(* IEC 61131-3 sources: TA/Tests/RetainTest/Man (part 21) *)

    RETAINTEST_AUTO_STRUCTUREARRAYARRAY.ARRAYARRAY_LREAL[2][0] := RETAINTEST_AUTO_STRUCTUREARRAYARRAY.ARRAYARRAY_LREAL[2][0] + 1.1;
    RETAINTEST_AUTO_STRUCTUREARRAYARRAY.ARRAYARRAY_LREAL[2][1] := RETAINTEST_AUTO_STRUCTUREARRAYARRAY.ARRAYARRAY_LREAL[2][1] + 1.1;
    RETAINTEST_AUTO_STRUCTUREARRAYARRAY.ARRAYARRAY_LREAL[2][2] := RETAINTEST_AUTO_STRUCTUREARRAYARRAY.ARRAYARRAY_LREAL[2][2] + 1.1;
    RETAINTEST_AUTO_STRUCTUREARRAYARRAY.ARRAYARRAY_LREAL[2][3] := RETAINTEST_AUTO_STRUCTUREARRAYARRAY.ARRAYARRAY_LREAL[2][3] + 1.1;
    RETAINTEST_AUTO_STRUCTUREARRAYARRAY.ARRAYARRAY_LREAL[2][4] := RETAINTEST_AUTO_STRUCTUREARRAYARRAY.ARRAYARRAY_LREAL[2][4] + 1.1;
    RETAINTEST_AUTO_STRUCTUREARRAYARRAY.ARRAYARRAY_LREAL[2][5] := RETAINTEST_AUTO_STRUCTUREARRAYARRAY.ARRAYARRAY_LREAL[2][5] + 1.1;
    RETAINTEST_AUTO_STRUCTUREARRAYARRAY.ARRAYARRAY_LREAL[2][6] := RETAINTEST_AUTO_STRUCTUREARRAYARRAY.ARRAYARRAY_LREAL[2][6] + 1.1;
    RETAINTEST_AUTO_STRUCTUREARRAYARRAY.ARRAYARRAY_LREAL[2][7] := RETAINTEST_AUTO_STRUCTUREARRAYARRAY.ARRAYARRAY_LREAL[2][7] + 1.1;
    RETAINTEST_AUTO_STRUCTUREARRAYARRAY.ARRAYARRAY_LREAL[2][8] := RETAINTEST_AUTO_STRUCTUREARRAYARRAY.ARRAYARRAY_LREAL[2][8] + 1.1;
    RETAINTEST_AUTO_STRUCTUREARRAYARRAY.ARRAYARRAY_LREAL[2][9] := RETAINTEST_AUTO_STRUCTUREARRAYARRAY.ARRAYARRAY_LREAL[2][9] + 1.1;

    RETAINTEST_AUTO_STRUCTUREARRAYARRAY.ARRAYARRAY_LREAL[3][0] := RETAINTEST_AUTO_STRUCTUREARRAYARRAY.ARRAYARRAY_LREAL[3][0] + 1.1;
    RETAINTEST_AUTO_STRUCTUREARRAYARRAY.ARRAYARRAY_LREAL[3][1] := RETAINTEST_AUTO_STRUCTUREARRAYARRAY.ARRAYARRAY_LREAL[3][1] + 1.1;
    RETAINTEST_AUTO_STRUCTUREARRAYARRAY.ARRAYARRAY_LREAL[3][2] := RETAINTEST_AUTO_STRUCTUREARRAYARRAY.ARRAYARRAY_LREAL[3][2] + 1.1;
    RETAINTEST_AUTO_STRUCTUREARRAYARRAY.ARRAYARRAY_LREAL[3][3] := RETAINTEST_AUTO_STRUCTUREARRAYARRAY.ARRAYARRAY_LREAL[3][3] + 1.1;
    RETAINTEST_AUTO_STRUCTUREARRAYARRAY.ARRAYARRAY_LREAL[3][4] := RETAINTEST_AUTO_STRUCTUREARRAYARRAY.ARRAYARRAY_LREAL[3][4] + 1.1;
    RETAINTEST_AUTO_STRUCTUREARRAYARRAY.ARRAYARRAY_LREAL[3][5] := RETAINTEST_AUTO_STRUCTUREARRAYARRAY.ARRAYARRAY_LREAL[3][5] + 1.1;
    RETAINTEST_AUTO_STRUCTUREARRAYARRAY.ARRAYARRAY_LREAL[3][6] := RETAINTEST_AUTO_STRUCTUREARRAYARRAY.ARRAYARRAY_LREAL[3][6] + 1.1;
    RETAINTEST_AUTO_STRUCTUREARRAYARRAY.ARRAYARRAY_LREAL[3][7] := RETAINTEST_AUTO_STRUCTUREARRAYARRAY.ARRAYARRAY_LREAL[3][7] + 1.1;
    RETAINTEST_AUTO_STRUCTUREARRAYARRAY.ARRAYARRAY_LREAL[3][8] := RETAINTEST_AUTO_STRUCTUREARRAYARRAY.ARRAYARRAY_LREAL[3][8] + 1.1;
    RETAINTEST_AUTO_STRUCTUREARRAYARRAY.ARRAYARRAY_LREAL[3][9] := RETAINTEST_AUTO_STRUCTUREARRAYARRAY.ARRAYARRAY_LREAL[3][9] + 1.1;

    RETAINTEST_AUTO_STRUCTUREARRAYARRAY.ARRAYARRAY_LREAL[4][0] := RETAINTEST_AUTO_STRUCTUREARRAYARRAY.ARRAYARRAY_LREAL[4][0] + 1.1;
    RETAINTEST_AUTO_STRUCTUREARRAYARRAY.ARRAYARRAY_LREAL[4][1] := RETAINTEST_AUTO_STRUCTUREARRAYARRAY.ARRAYARRAY_LREAL[4][1] + 1.1;
    RETAINTEST_AUTO_STRUCTUREARRAYARRAY.ARRAYARRAY_LREAL[4][2] := RETAINTEST_AUTO_STRUCTUREARRAYARRAY.ARRAYARRAY_LREAL[4][2] + 1.1;
    RETAINTEST_AUTO_STRUCTUREARRAYARRAY.ARRAYARRAY_LREAL[4][3] := RETAINTEST_AUTO_STRUCTUREARRAYARRAY.ARRAYARRAY_LREAL[4][3] + 1.1;
    RETAINTEST_AUTO_STRUCTUREARRAYARRAY.ARRAYARRAY_LREAL[4][4] := RETAINTEST_AUTO_STRUCTUREARRAYARRAY.ARRAYARRAY_LREAL[4][4] + 1.1;
    RETAINTEST_AUTO_STRUCTUREARRAYARRAY.ARRAYARRAY_LREAL[4][5] := RETAINTEST_AUTO_STRUCTUREARRAYARRAY.ARRAYARRAY_LREAL[4][5] + 1.1;
    RETAINTEST_AUTO_STRUCTUREARRAYARRAY.ARRAYARRAY_LREAL[4][6] := RETAINTEST_AUTO_STRUCTUREARRAYARRAY.ARRAYARRAY_LREAL[4][6] + 1.1;
    RETAINTEST_AUTO_STRUCTUREARRAYARRAY.ARRAYARRAY_LREAL[4][7] := RETAINTEST_AUTO_STRUCTUREARRAYARRAY.ARRAYARRAY_LREAL[4][7] + 1.1;
    RETAINTEST_AUTO_STRUCTUREARRAYARRAY.ARRAYARRAY_LREAL[4][8] := RETAINTEST_AUTO_STRUCTUREARRAYARRAY.ARRAYARRAY_LREAL[4][8] + 1.1;
    RETAINTEST_AUTO_STRUCTUREARRAYARRAY.ARRAYARRAY_LREAL[4][9] := RETAINTEST_AUTO_STRUCTUREARRAYARRAY.ARRAYARRAY_LREAL[4][9] + 1.1;

    RETAINTEST_AUTO_STRUCTUREARRAYARRAY.ARRAYARRAY_LREAL[5][0] := RETAINTEST_AUTO_STRUCTUREARRAYARRAY.ARRAYARRAY_LREAL[5][0] + 1.1;
    RETAINTEST_AUTO_STRUCTUREARRAYARRAY.ARRAYARRAY_LREAL[5][1] := RETAINTEST_AUTO_STRUCTUREARRAYARRAY.ARRAYARRAY_LREAL[5][1] + 1.1;
    RETAINTEST_AUTO_STRUCTUREARRAYARRAY.ARRAYARRAY_LREAL[5][2] := RETAINTEST_AUTO_STRUCTUREARRAYARRAY.ARRAYARRAY_LREAL[5][2] + 1.1;
    RETAINTEST_AUTO_STRUCTUREARRAYARRAY.ARRAYARRAY_LREAL[5][3] := RETAINTEST_AUTO_STRUCTUREARRAYARRAY.ARRAYARRAY_LREAL[5][3] + 1.1;
    RETAINTEST_AUTO_STRUCTUREARRAYARRAY.ARRAYARRAY_LREAL[5][4] := RETAINTEST_AUTO_STRUCTUREARRAYARRAY.ARRAYARRAY_LREAL[5][4] + 1.1;
    RETAINTEST_AUTO_STRUCTUREARRAYARRAY.ARRAYARRAY_LREAL[5][5] := RETAINTEST_AUTO_STRUCTUREARRAYARRAY.ARRAYARRAY_LREAL[5][5] + 1.1;
    RETAINTEST_AUTO_STRUCTUREARRAYARRAY.ARRAYARRAY_LREAL[5][6] := RETAINTEST_AUTO_STRUCTUREARRAYARRAY.ARRAYARRAY_LREAL[5][6] + 1.1;
    RETAINTEST_AUTO_STRUCTUREARRAYARRAY.ARRAYARRAY_LREAL[5][7] := RETAINTEST_AUTO_STRUCTUREARRAYARRAY.ARRAYARRAY_LREAL[5][7] + 1.1;
    RETAINTEST_AUTO_STRUCTUREARRAYARRAY.ARRAYARRAY_LREAL[5][8] := RETAINTEST_AUTO_STRUCTUREARRAYARRAY.ARRAYARRAY_LREAL[5][8] + 1.1;
    RETAINTEST_AUTO_STRUCTUREARRAYARRAY.ARRAYARRAY_LREAL[5][9] := RETAINTEST_AUTO_STRUCTUREARRAYARRAY.ARRAYARRAY_LREAL[5][9] + 1.1;

    RETAINTEST_AUTO_STRUCTUREARRAYARRAY.ARRAYARRAY_LREAL[6][0] := RETAINTEST_AUTO_STRUCTUREARRAYARRAY.ARRAYARRAY_LREAL[6][0] + 1.1;
    RETAINTEST_AUTO_STRUCTUREARRAYARRAY.ARRAYARRAY_LREAL[6][1] := RETAINTEST_AUTO_STRUCTUREARRAYARRAY.ARRAYARRAY_LREAL[6][1] + 1.1;
    RETAINTEST_AUTO_STRUCTUREARRAYARRAY.ARRAYARRAY_LREAL[6][2] := RETAINTEST_AUTO_STRUCTUREARRAYARRAY.ARRAYARRAY_LREAL[6][2] + 1.1;
    RETAINTEST_AUTO_STRUCTUREARRAYARRAY.ARRAYARRAY_LREAL[6][3] := RETAINTEST_AUTO_STRUCTUREARRAYARRAY.ARRAYARRAY_LREAL[6][3] + 1.1;
    RETAINTEST_AUTO_STRUCTUREARRAYARRAY.ARRAYARRAY_LREAL[6][4] := RETAINTEST_AUTO_STRUCTUREARRAYARRAY.ARRAYARRAY_LREAL[6][4] + 1.1;
    RETAINTEST_AUTO_STRUCTUREARRAYARRAY.ARRAYARRAY_LREAL[6][5] := RETAINTEST_AUTO_STRUCTUREARRAYARRAY.ARRAYARRAY_LREAL[6][5] + 1.1;
    RETAINTEST_AUTO_STRUCTUREARRAYARRAY.ARRAYARRAY_LREAL[6][6] := RETAINTEST_AUTO_STRUCTUREARRAYARRAY.ARRAYARRAY_LREAL[6][6] + 1.1;
    RETAINTEST_AUTO_STRUCTUREARRAYARRAY.ARRAYARRAY_LREAL[6][7] := RETAINTEST_AUTO_STRUCTUREARRAYARRAY.ARRAYARRAY_LREAL[6][7] + 1.1;
    RETAINTEST_AUTO_STRUCTUREARRAYARRAY.ARRAYARRAY_LREAL[6][8] := RETAINTEST_AUTO_STRUCTUREARRAYARRAY.ARRAYARRAY_LREAL[6][8] + 1.1;
    RETAINTEST_AUTO_STRUCTUREARRAYARRAY.ARRAYARRAY_LREAL[6][9] := RETAINTEST_AUTO_STRUCTUREARRAYARRAY.ARRAYARRAY_LREAL[6][9] + 1.1;

    RETAINTEST_AUTO_STRUCTUREARRAYARRAY.ARRAYARRAY_LREAL[7][0] := RETAINTEST_AUTO_STRUCTUREARRAYARRAY.ARRAYARRAY_LREAL[6][0];
    RETAINTEST_AUTO_STRUCTUREARRAYARRAY.ARRAYARRAY_LREAL[7][1] := RETAINTEST_AUTO_STRUCTUREARRAYARRAY.ARRAYARRAY_LREAL[6][1];
    RETAINTEST_AUTO_STRUCTUREARRAYARRAY.ARRAYARRAY_LREAL[7][2] := RETAINTEST_AUTO_STRUCTUREARRAYARRAY.ARRAYARRAY_LREAL[6][2];
    RETAINTEST_AUTO_STRUCTUREARRAYARRAY.ARRAYARRAY_LREAL[7][3] := RETAINTEST_AUTO_STRUCTUREARRAYARRAY.ARRAYARRAY_LREAL[6][3];
    RETAINTEST_AUTO_STRUCTUREARRAYARRAY.ARRAYARRAY_LREAL[7][4] := RETAINTEST_AUTO_STRUCTUREARRAYARRAY.ARRAYARRAY_LREAL[6][4];
    RETAINTEST_AUTO_STRUCTUREARRAYARRAY.ARRAYARRAY_LREAL[7][5] := RETAINTEST_AUTO_STRUCTUREARRAYARRAY.ARRAYARRAY_LREAL[6][5];
    RETAINTEST_AUTO_STRUCTUREARRAYARRAY.ARRAYARRAY_LREAL[7][6] := RETAINTEST_AUTO_STRUCTUREARRAYARRAY.ARRAYARRAY_LREAL[6][6];
    RETAINTEST_AUTO_STRUCTUREARRAYARRAY.ARRAYARRAY_LREAL[7][7] := RETAINTEST_AUTO_STRUCTUREARRAYARRAY.ARRAYARRAY_LREAL[6][7];
    RETAINTEST_AUTO_STRUCTUREARRAYARRAY.ARRAYARRAY_LREAL[7][8] := RETAINTEST_AUTO_STRUCTUREARRAYARRAY.ARRAYARRAY_LREAL[6][8];
    RETAINTEST_AUTO_STRUCTUREARRAYARRAY.ARRAYARRAY_LREAL[7][9] := RETAINTEST_AUTO_STRUCTUREARRAYARRAY.ARRAYARRAY_LREAL[6][9];

    RETAINTEST_AUTO_STRUCTUREARRAYARRAY.ARRAYARRAY_LWORD[0][0] := RETAINTEST_AUTO_STRUCTUREARRAYARRAY.ARRAYARRAY_LWORD[0][0] + 1;
    RETAINTEST_AUTO_STRUCTUREARRAYARRAY.ARRAYARRAY_LWORD[0][1] := RETAINTEST_AUTO_STRUCTUREARRAYARRAY.ARRAYARRAY_LWORD[0][1] + 1;
    RETAINTEST_AUTO_STRUCTUREARRAYARRAY.ARRAYARRAY_LWORD[0][2] := RETAINTEST_AUTO_STRUCTUREARRAYARRAY.ARRAYARRAY_LWORD[0][2] + 1;
    RETAINTEST_AUTO_STRUCTUREARRAYARRAY.ARRAYARRAY_LWORD[0][3] := RETAINTEST_AUTO_STRUCTUREARRAYARRAY.ARRAYARRAY_LWORD[0][3] + 1;
    RETAINTEST_AUTO_STRUCTUREARRAYARRAY.ARRAYARRAY_LWORD[0][4] := RETAINTEST_AUTO_STRUCTUREARRAYARRAY.ARRAYARRAY_LWORD[0][4] + 1;
    RETAINTEST_AUTO_STRUCTUREARRAYARRAY.ARRAYARRAY_LWORD[0][5] := RETAINTEST_AUTO_STRUCTUREARRAYARRAY.ARRAYARRAY_LWORD[0][5] + 1;
    RETAINTEST_AUTO_STRUCTUREARRAYARRAY.ARRAYARRAY_LWORD[0][6] := RETAINTEST_AUTO_STRUCTUREARRAYARRAY.ARRAYARRAY_LWORD[0][6] + 1;
    RETAINTEST_AUTO_STRUCTUREARRAYARRAY.ARRAYARRAY_LWORD[0][7] := RETAINTEST_AUTO_STRUCTUREARRAYARRAY.ARRAYARRAY_LWORD[0][7] + 1;
    RETAINTEST_AUTO_STRUCTUREARRAYARRAY.ARRAYARRAY_LWORD[0][8] := RETAINTEST_AUTO_STRUCTUREARRAYARRAY.ARRAYARRAY_LWORD[0][6];
    RETAINTEST_AUTO_STRUCTUREARRAYARRAY.ARRAYARRAY_LWORD[0][9] := RETAINTEST_AUTO_STRUCTUREARRAYARRAY.ARRAYARRAY_LWORD[0][7];

    RETAINTEST_AUTO_STRUCTUREARRAYARRAY.ARRAYARRAY_LWORD[1][0] := RETAINTEST_AUTO_STRUCTUREARRAYARRAY.ARRAYARRAY_LWORD[1][0] + 1;
    RETAINTEST_AUTO_STRUCTUREARRAYARRAY.ARRAYARRAY_LWORD[1][1] := RETAINTEST_AUTO_STRUCTUREARRAYARRAY.ARRAYARRAY_LWORD[1][1] + 1;
    RETAINTEST_AUTO_STRUCTUREARRAYARRAY.ARRAYARRAY_LWORD[1][2] := RETAINTEST_AUTO_STRUCTUREARRAYARRAY.ARRAYARRAY_LWORD[1][2] + 1;
    RETAINTEST_AUTO_STRUCTUREARRAYARRAY.ARRAYARRAY_LWORD[1][3] := RETAINTEST_AUTO_STRUCTUREARRAYARRAY.ARRAYARRAY_LWORD[1][3] + 1;
    RETAINTEST_AUTO_STRUCTUREARRAYARRAY.ARRAYARRAY_LWORD[1][4] := RETAINTEST_AUTO_STRUCTUREARRAYARRAY.ARRAYARRAY_LWORD[1][4] + 1;
    RETAINTEST_AUTO_STRUCTUREARRAYARRAY.ARRAYARRAY_LWORD[1][5] := RETAINTEST_AUTO_STRUCTUREARRAYARRAY.ARRAYARRAY_LWORD[1][5] + 1;
    RETAINTEST_AUTO_STRUCTUREARRAYARRAY.ARRAYARRAY_LWORD[1][6] := RETAINTEST_AUTO_STRUCTUREARRAYARRAY.ARRAYARRAY_LWORD[1][6] + 1;
    RETAINTEST_AUTO_STRUCTUREARRAYARRAY.ARRAYARRAY_LWORD[1][7] := RETAINTEST_AUTO_STRUCTUREARRAYARRAY.ARRAYARRAY_LWORD[1][7] + 1;
    RETAINTEST_AUTO_STRUCTUREARRAYARRAY.ARRAYARRAY_LWORD[1][8] := RETAINTEST_AUTO_STRUCTUREARRAYARRAY.ARRAYARRAY_LWORD[1][6];
    RETAINTEST_AUTO_STRUCTUREARRAYARRAY.ARRAYARRAY_LWORD[1][9] := RETAINTEST_AUTO_STRUCTUREARRAYARRAY.ARRAYARRAY_LWORD[1][7];

    RETAINTEST_AUTO_STRUCTUREARRAYARRAY.ARRAYARRAY_LWORD[2][0] := RETAINTEST_AUTO_STRUCTUREARRAYARRAY.ARRAYARRAY_LWORD[2][0] + 1;
    RETAINTEST_AUTO_STRUCTUREARRAYARRAY.ARRAYARRAY_LWORD[2][1] := RETAINTEST_AUTO_STRUCTUREARRAYARRAY.ARRAYARRAY_LWORD[2][1] + 1;
    RETAINTEST_AUTO_STRUCTUREARRAYARRAY.ARRAYARRAY_LWORD[2][2] := RETAINTEST_AUTO_STRUCTUREARRAYARRAY.ARRAYARRAY_LWORD[2][2] + 1;
    RETAINTEST_AUTO_STRUCTUREARRAYARRAY.ARRAYARRAY_LWORD[2][3] := RETAINTEST_AUTO_STRUCTUREARRAYARRAY.ARRAYARRAY_LWORD[2][3] + 1;
    RETAINTEST_AUTO_STRUCTUREARRAYARRAY.ARRAYARRAY_LWORD[2][4] := RETAINTEST_AUTO_STRUCTUREARRAYARRAY.ARRAYARRAY_LWORD[2][4] + 1;
    RETAINTEST_AUTO_STRUCTUREARRAYARRAY.ARRAYARRAY_LWORD[2][5] := RETAINTEST_AUTO_STRUCTUREARRAYARRAY.ARRAYARRAY_LWORD[2][5] + 1;
    RETAINTEST_AUTO_STRUCTUREARRAYARRAY.ARRAYARRAY_LWORD[2][6] := RETAINTEST_AUTO_STRUCTUREARRAYARRAY.ARRAYARRAY_LWORD[2][6] + 1;
    RETAINTEST_AUTO_STRUCTUREARRAYARRAY.ARRAYARRAY_LWORD[2][7] := RETAINTEST_AUTO_STRUCTUREARRAYARRAY.ARRAYARRAY_LWORD[2][7] + 1;
    RETAINTEST_AUTO_STRUCTUREARRAYARRAY.ARRAYARRAY_LWORD[2][8] := RETAINTEST_AUTO_STRUCTUREARRAYARRAY.ARRAYARRAY_LWORD[2][8] + 1;
    RETAINTEST_AUTO_STRUCTUREARRAYARRAY.ARRAYARRAY_LWORD[2][9] := RETAINTEST_AUTO_STRUCTUREARRAYARRAY.ARRAYARRAY_LWORD[2][9] + 1;

    RETAINTEST_AUTO_STRUCTUREARRAYARRAY.ARRAYARRAY_LWORD[3][0] := RETAINTEST_AUTO_STRUCTUREARRAYARRAY.ARRAYARRAY_LWORD[3][0] + 1;
    RETAINTEST_AUTO_STRUCTUREARRAYARRAY.ARRAYARRAY_LWORD[3][1] := RETAINTEST_AUTO_STRUCTUREARRAYARRAY.ARRAYARRAY_LWORD[3][1] + 1;
    RETAINTEST_AUTO_STRUCTUREARRAYARRAY.ARRAYARRAY_LWORD[3][2] := RETAINTEST_AUTO_STRUCTUREARRAYARRAY.ARRAYARRAY_LWORD[3][2] + 1;
    RETAINTEST_AUTO_STRUCTUREARRAYARRAY.ARRAYARRAY_LWORD[3][3] := RETAINTEST_AUTO_STRUCTUREARRAYARRAY.ARRAYARRAY_LWORD[3][3] + 1;
    RETAINTEST_AUTO_STRUCTUREARRAYARRAY.ARRAYARRAY_LWORD[3][4] := RETAINTEST_AUTO_STRUCTUREARRAYARRAY.ARRAYARRAY_LWORD[3][4] + 1;
    RETAINTEST_AUTO_STRUCTUREARRAYARRAY.ARRAYARRAY_LWORD[3][5] := RETAINTEST_AUTO_STRUCTUREARRAYARRAY.ARRAYARRAY_LWORD[3][5] + 1;
    RETAINTEST_AUTO_STRUCTUREARRAYARRAY.ARRAYARRAY_LWORD[3][6] := RETAINTEST_AUTO_STRUCTUREARRAYARRAY.ARRAYARRAY_LWORD[3][6] + 1;
    RETAINTEST_AUTO_STRUCTUREARRAYARRAY.ARRAYARRAY_LWORD[3][7] := RETAINTEST_AUTO_STRUCTUREARRAYARRAY.ARRAYARRAY_LWORD[3][7] + 1;
    RETAINTEST_AUTO_STRUCTUREARRAYARRAY.ARRAYARRAY_LWORD[3][8] := RETAINTEST_AUTO_STRUCTUREARRAYARRAY.ARRAYARRAY_LWORD[3][8] + 1;
    RETAINTEST_AUTO_STRUCTUREARRAYARRAY.ARRAYARRAY_LWORD[3][9] := RETAINTEST_AUTO_STRUCTUREARRAYARRAY.ARRAYARRAY_LWORD[3][9] + 1;

    RETAINTEST_AUTO_STRUCTUREARRAYARRAY.ARRAYARRAY_LWORD[4][0] := RETAINTEST_AUTO_STRUCTUREARRAYARRAY.ARRAYARRAY_LWORD[4][0] + 1;
    RETAINTEST_AUTO_STRUCTUREARRAYARRAY.ARRAYARRAY_LWORD[4][1] := RETAINTEST_AUTO_STRUCTUREARRAYARRAY.ARRAYARRAY_LWORD[4][1] + 1;
    RETAINTEST_AUTO_STRUCTUREARRAYARRAY.ARRAYARRAY_LWORD[4][2] := RETAINTEST_AUTO_STRUCTUREARRAYARRAY.ARRAYARRAY_LWORD[4][2] + 1;
    RETAINTEST_AUTO_STRUCTUREARRAYARRAY.ARRAYARRAY_LWORD[4][3] := RETAINTEST_AUTO_STRUCTUREARRAYARRAY.ARRAYARRAY_LWORD[4][3] + 1;
    RETAINTEST_AUTO_STRUCTUREARRAYARRAY.ARRAYARRAY_LWORD[4][4] := RETAINTEST_AUTO_STRUCTUREARRAYARRAY.ARRAYARRAY_LWORD[4][4] + 1;
    RETAINTEST_AUTO_STRUCTUREARRAYARRAY.ARRAYARRAY_LWORD[4][5] := RETAINTEST_AUTO_STRUCTUREARRAYARRAY.ARRAYARRAY_LWORD[4][5] + 1;
    RETAINTEST_AUTO_STRUCTUREARRAYARRAY.ARRAYARRAY_LWORD[4][6] := RETAINTEST_AUTO_STRUCTUREARRAYARRAY.ARRAYARRAY_LWORD[4][6] + 1;
    RETAINTEST_AUTO_STRUCTUREARRAYARRAY.ARRAYARRAY_LWORD[4][7] := RETAINTEST_AUTO_STRUCTUREARRAYARRAY.ARRAYARRAY_LWORD[4][7] + 1;
    RETAINTEST_AUTO_STRUCTUREARRAYARRAY.ARRAYARRAY_LWORD[4][8] := RETAINTEST_AUTO_STRUCTUREARRAYARRAY.ARRAYARRAY_LWORD[4][8] + 1;
    RETAINTEST_AUTO_STRUCTUREARRAYARRAY.ARRAYARRAY_LWORD[4][9] := RETAINTEST_AUTO_STRUCTUREARRAYARRAY.ARRAYARRAY_LWORD[4][9] + 1;

    RETAINTEST_AUTO_STRUCTUREARRAYARRAY.ARRAYARRAY_LWORD[5][0] := RETAINTEST_AUTO_STRUCTUREARRAYARRAY.ARRAYARRAY_LWORD[5][0] + 1;
    RETAINTEST_AUTO_STRUCTUREARRAYARRAY.ARRAYARRAY_LWORD[5][1] := RETAINTEST_AUTO_STRUCTUREARRAYARRAY.ARRAYARRAY_LWORD[5][1] + 1;
    RETAINTEST_AUTO_STRUCTUREARRAYARRAY.ARRAYARRAY_LWORD[5][2] := RETAINTEST_AUTO_STRUCTUREARRAYARRAY.ARRAYARRAY_LWORD[5][2] + 1;
    RETAINTEST_AUTO_STRUCTUREARRAYARRAY.ARRAYARRAY_LWORD[5][3] := RETAINTEST_AUTO_STRUCTUREARRAYARRAY.ARRAYARRAY_LWORD[5][3] + 1;
    RETAINTEST_AUTO_STRUCTUREARRAYARRAY.ARRAYARRAY_LWORD[5][4] := RETAINTEST_AUTO_STRUCTUREARRAYARRAY.ARRAYARRAY_LWORD[5][4] + 1;
    RETAINTEST_AUTO_STRUCTUREARRAYARRAY.ARRAYARRAY_LWORD[5][5] := RETAINTEST_AUTO_STRUCTUREARRAYARRAY.ARRAYARRAY_LWORD[5][5] + 1;
    RETAINTEST_AUTO_STRUCTUREARRAYARRAY.ARRAYARRAY_LWORD[5][6] := RETAINTEST_AUTO_STRUCTUREARRAYARRAY.ARRAYARRAY_LWORD[5][6] + 1;
    RETAINTEST_AUTO_STRUCTUREARRAYARRAY.ARRAYARRAY_LWORD[5][7] := RETAINTEST_AUTO_STRUCTUREARRAYARRAY.ARRAYARRAY_LWORD[5][7] + 1;
    RETAINTEST_AUTO_STRUCTUREARRAYARRAY.ARRAYARRAY_LWORD[5][8] := RETAINTEST_AUTO_STRUCTUREARRAYARRAY.ARRAYARRAY_LWORD[5][8] + 1;
    RETAINTEST_AUTO_STRUCTUREARRAYARRAY.ARRAYARRAY_LWORD[5][9] := RETAINTEST_AUTO_STRUCTUREARRAYARRAY.ARRAYARRAY_LWORD[5][9] + 1;

    RETAINTEST_AUTO_STRUCTUREARRAYARRAY.ARRAYARRAY_LWORD[6][0] := RETAINTEST_AUTO_STRUCTUREARRAYARRAY.ARRAYARRAY_LWORD[6][0] + 1;
    RETAINTEST_AUTO_STRUCTUREARRAYARRAY.ARRAYARRAY_LWORD[6][1] := RETAINTEST_AUTO_STRUCTUREARRAYARRAY.ARRAYARRAY_LWORD[6][1] + 1;
    RETAINTEST_AUTO_STRUCTUREARRAYARRAY.ARRAYARRAY_LWORD[6][2] := RETAINTEST_AUTO_STRUCTUREARRAYARRAY.ARRAYARRAY_LWORD[6][2] + 1;
    RETAINTEST_AUTO_STRUCTUREARRAYARRAY.ARRAYARRAY_LWORD[6][3] := RETAINTEST_AUTO_STRUCTUREARRAYARRAY.ARRAYARRAY_LWORD[6][3] + 1;
    RETAINTEST_AUTO_STRUCTUREARRAYARRAY.ARRAYARRAY_LWORD[6][4] := RETAINTEST_AUTO_STRUCTUREARRAYARRAY.ARRAYARRAY_LWORD[6][4] + 1;
    RETAINTEST_AUTO_STRUCTUREARRAYARRAY.ARRAYARRAY_LWORD[6][5] := RETAINTEST_AUTO_STRUCTUREARRAYARRAY.ARRAYARRAY_LWORD[6][5] + 1;
    RETAINTEST_AUTO_STRUCTUREARRAYARRAY.ARRAYARRAY_LWORD[6][6] := RETAINTEST_AUTO_STRUCTUREARRAYARRAY.ARRAYARRAY_LWORD[6][6] + 1;
    RETAINTEST_AUTO_STRUCTUREARRAYARRAY.ARRAYARRAY_LWORD[6][7] := RETAINTEST_AUTO_STRUCTUREARRAYARRAY.ARRAYARRAY_LWORD[6][7] + 1;
    RETAINTEST_AUTO_STRUCTUREARRAYARRAY.ARRAYARRAY_LWORD[6][8] := RETAINTEST_AUTO_STRUCTUREARRAYARRAY.ARRAYARRAY_LWORD[6][8] + 1;
    RETAINTEST_AUTO_STRUCTUREARRAYARRAY.ARRAYARRAY_LWORD[6][9] := RETAINTEST_AUTO_STRUCTUREARRAYARRAY.ARRAYARRAY_LWORD[6][9] + 1;

    RETAINTEST_AUTO_STRUCTUREARRAYARRAY.ARRAYARRAY_LWORD[7][0] := RETAINTEST_AUTO_STRUCTUREARRAYARRAY.ARRAYARRAY_LWORD[6][0];
    RETAINTEST_AUTO_STRUCTUREARRAYARRAY.ARRAYARRAY_LWORD[7][1] := RETAINTEST_AUTO_STRUCTUREARRAYARRAY.ARRAYARRAY_LWORD[6][1];
    RETAINTEST_AUTO_STRUCTUREARRAYARRAY.ARRAYARRAY_LWORD[7][2] := RETAINTEST_AUTO_STRUCTUREARRAYARRAY.ARRAYARRAY_LWORD[6][2];
    RETAINTEST_AUTO_STRUCTUREARRAYARRAY.ARRAYARRAY_LWORD[7][3] := RETAINTEST_AUTO_STRUCTUREARRAYARRAY.ARRAYARRAY_LWORD[6][3];
    RETAINTEST_AUTO_STRUCTUREARRAYARRAY.ARRAYARRAY_LWORD[7][4] := RETAINTEST_AUTO_STRUCTUREARRAYARRAY.ARRAYARRAY_LWORD[6][4];
    RETAINTEST_AUTO_STRUCTUREARRAYARRAY.ARRAYARRAY_LWORD[7][5] := RETAINTEST_AUTO_STRUCTUREARRAYARRAY.ARRAYARRAY_LWORD[6][5];
    RETAINTEST_AUTO_STRUCTUREARRAYARRAY.ARRAYARRAY_LWORD[7][6] := RETAINTEST_AUTO_STRUCTUREARRAYARRAY.ARRAYARRAY_LWORD[6][6];
    RETAINTEST_AUTO_STRUCTUREARRAYARRAY.ARRAYARRAY_LWORD[7][7] := RETAINTEST_AUTO_STRUCTUREARRAYARRAY.ARRAYARRAY_LWORD[6][7];
    RETAINTEST_AUTO_STRUCTUREARRAYARRAY.ARRAYARRAY_LWORD[7][8] := RETAINTEST_AUTO_STRUCTUREARRAYARRAY.ARRAYARRAY_LWORD[6][8];
    RETAINTEST_AUTO_STRUCTUREARRAYARRAY.ARRAYARRAY_LWORD[7][9] := RETAINTEST_AUTO_STRUCTUREARRAYARRAY.ARRAYARRAY_LWORD[6][9];

    RETAINTEST_AUTO_STRUCTUREARRAYARRAY.ARRAYARRAY_REAL[0][0] := RETAINTEST_AUTO_STRUCTUREARRAYARRAY.ARRAYARRAY_REAL[0][0] + 1.1;
    RETAINTEST_AUTO_STRUCTUREARRAYARRAY.ARRAYARRAY_REAL[0][1] := RETAINTEST_AUTO_STRUCTUREARRAYARRAY.ARRAYARRAY_REAL[0][1] + 1.1;
    RETAINTEST_AUTO_STRUCTUREARRAYARRAY.ARRAYARRAY_REAL[0][2] := RETAINTEST_AUTO_STRUCTUREARRAYARRAY.ARRAYARRAY_REAL[0][2] + 1.1;
    RETAINTEST_AUTO_STRUCTUREARRAYARRAY.ARRAYARRAY_REAL[0][3] := RETAINTEST_AUTO_STRUCTUREARRAYARRAY.ARRAYARRAY_REAL[0][3] + 1.1;
    RETAINTEST_AUTO_STRUCTUREARRAYARRAY.ARRAYARRAY_REAL[0][4] := RETAINTEST_AUTO_STRUCTUREARRAYARRAY.ARRAYARRAY_REAL[0][4] + 1.1;
    RETAINTEST_AUTO_STRUCTUREARRAYARRAY.ARRAYARRAY_REAL[0][5] := RETAINTEST_AUTO_STRUCTUREARRAYARRAY.ARRAYARRAY_REAL[0][5] + 1.1;
    RETAINTEST_AUTO_STRUCTUREARRAYARRAY.ARRAYARRAY_REAL[0][6] := RETAINTEST_AUTO_STRUCTUREARRAYARRAY.ARRAYARRAY_REAL[0][6] + 1.1;
    RETAINTEST_AUTO_STRUCTUREARRAYARRAY.ARRAYARRAY_REAL[0][7] := RETAINTEST_AUTO_STRUCTUREARRAYARRAY.ARRAYARRAY_REAL[0][7] + 1.1;
    RETAINTEST_AUTO_STRUCTUREARRAYARRAY.ARRAYARRAY_REAL[0][8] := RETAINTEST_AUTO_STRUCTUREARRAYARRAY.ARRAYARRAY_REAL[0][6];
    RETAINTEST_AUTO_STRUCTUREARRAYARRAY.ARRAYARRAY_REAL[0][9] := RETAINTEST_AUTO_STRUCTUREARRAYARRAY.ARRAYARRAY_REAL[0][7];

    RETAINTEST_AUTO_STRUCTUREARRAYARRAY.ARRAYARRAY_REAL[1][0] := RETAINTEST_AUTO_STRUCTUREARRAYARRAY.ARRAYARRAY_REAL[1][0] + 1.1;
    RETAINTEST_AUTO_STRUCTUREARRAYARRAY.ARRAYARRAY_REAL[1][1] := RETAINTEST_AUTO_STRUCTUREARRAYARRAY.ARRAYARRAY_REAL[1][1] + 1.1;
    RETAINTEST_AUTO_STRUCTUREARRAYARRAY.ARRAYARRAY_REAL[1][2] := RETAINTEST_AUTO_STRUCTUREARRAYARRAY.ARRAYARRAY_REAL[1][2] + 1.1;
    RETAINTEST_AUTO_STRUCTUREARRAYARRAY.ARRAYARRAY_REAL[1][3] := RETAINTEST_AUTO_STRUCTUREARRAYARRAY.ARRAYARRAY_REAL[1][3] + 1.1;
    RETAINTEST_AUTO_STRUCTUREARRAYARRAY.ARRAYARRAY_REAL[1][4] := RETAINTEST_AUTO_STRUCTUREARRAYARRAY.ARRAYARRAY_REAL[1][4] + 1.1;
    RETAINTEST_AUTO_STRUCTUREARRAYARRAY.ARRAYARRAY_REAL[1][5] := RETAINTEST_AUTO_STRUCTUREARRAYARRAY.ARRAYARRAY_REAL[1][5] + 1.1;
    RETAINTEST_AUTO_STRUCTUREARRAYARRAY.ARRAYARRAY_REAL[1][6] := RETAINTEST_AUTO_STRUCTUREARRAYARRAY.ARRAYARRAY_REAL[1][6] + 1.1;
    RETAINTEST_AUTO_STRUCTUREARRAYARRAY.ARRAYARRAY_REAL[1][7] := RETAINTEST_AUTO_STRUCTUREARRAYARRAY.ARRAYARRAY_REAL[1][7] + 1.1;
    RETAINTEST_AUTO_STRUCTUREARRAYARRAY.ARRAYARRAY_REAL[1][8] := RETAINTEST_AUTO_STRUCTUREARRAYARRAY.ARRAYARRAY_REAL[1][6];
    RETAINTEST_AUTO_STRUCTUREARRAYARRAY.ARRAYARRAY_REAL[1][9] := RETAINTEST_AUTO_STRUCTUREARRAYARRAY.ARRAYARRAY_REAL[1][7];

    RETAINTEST_AUTO_STRUCTUREARRAYARRAY.ARRAYARRAY_REAL[2][0] := RETAINTEST_AUTO_STRUCTUREARRAYARRAY.ARRAYARRAY_REAL[2][0] + 1.1;
    RETAINTEST_AUTO_STRUCTUREARRAYARRAY.ARRAYARRAY_REAL[2][1] := RETAINTEST_AUTO_STRUCTUREARRAYARRAY.ARRAYARRAY_REAL[2][1] + 1.1;
    RETAINTEST_AUTO_STRUCTUREARRAYARRAY.ARRAYARRAY_REAL[2][2] := RETAINTEST_AUTO_STRUCTUREARRAYARRAY.ARRAYARRAY_REAL[2][2] + 1.1;
    RETAINTEST_AUTO_STRUCTUREARRAYARRAY.ARRAYARRAY_REAL[2][3] := RETAINTEST_AUTO_STRUCTUREARRAYARRAY.ARRAYARRAY_REAL[2][3] + 1.1;
    RETAINTEST_AUTO_STRUCTUREARRAYARRAY.ARRAYARRAY_REAL[2][4] := RETAINTEST_AUTO_STRUCTUREARRAYARRAY.ARRAYARRAY_REAL[2][4] + 1.1;
    RETAINTEST_AUTO_STRUCTUREARRAYARRAY.ARRAYARRAY_REAL[2][5] := RETAINTEST_AUTO_STRUCTUREARRAYARRAY.ARRAYARRAY_REAL[2][5] + 1.1;
    RETAINTEST_AUTO_STRUCTUREARRAYARRAY.ARRAYARRAY_REAL[2][6] := RETAINTEST_AUTO_STRUCTUREARRAYARRAY.ARRAYARRAY_REAL[2][6] + 1.1;
    RETAINTEST_AUTO_STRUCTUREARRAYARRAY.ARRAYARRAY_REAL[2][7] := RETAINTEST_AUTO_STRUCTUREARRAYARRAY.ARRAYARRAY_REAL[2][7] + 1.1;
    RETAINTEST_AUTO_STRUCTUREARRAYARRAY.ARRAYARRAY_REAL[2][8] := RETAINTEST_AUTO_STRUCTUREARRAYARRAY.ARRAYARRAY_REAL[2][8] + 1.1;
    RETAINTEST_AUTO_STRUCTUREARRAYARRAY.ARRAYARRAY_REAL[2][9] := RETAINTEST_AUTO_STRUCTUREARRAYARRAY.ARRAYARRAY_REAL[2][9] + 1.1;

    RETAINTEST_AUTO_STRUCTUREARRAYARRAY.ARRAYARRAY_REAL[3][0] := RETAINTEST_AUTO_STRUCTUREARRAYARRAY.ARRAYARRAY_REAL[3][0] + 1.1;
    RETAINTEST_AUTO_STRUCTUREARRAYARRAY.ARRAYARRAY_REAL[3][1] := RETAINTEST_AUTO_STRUCTUREARRAYARRAY.ARRAYARRAY_REAL[3][1] + 1.1;
    RETAINTEST_AUTO_STRUCTUREARRAYARRAY.ARRAYARRAY_REAL[3][2] := RETAINTEST_AUTO_STRUCTUREARRAYARRAY.ARRAYARRAY_REAL[3][2] + 1.1;
    RETAINTEST_AUTO_STRUCTUREARRAYARRAY.ARRAYARRAY_REAL[3][3] := RETAINTEST_AUTO_STRUCTUREARRAYARRAY.ARRAYARRAY_REAL[3][3] + 1.1;
    RETAINTEST_AUTO_STRUCTUREARRAYARRAY.ARRAYARRAY_REAL[3][4] := RETAINTEST_AUTO_STRUCTUREARRAYARRAY.ARRAYARRAY_REAL[3][4] + 1.1;
    RETAINTEST_AUTO_STRUCTUREARRAYARRAY.ARRAYARRAY_REAL[3][5] := RETAINTEST_AUTO_STRUCTUREARRAYARRAY.ARRAYARRAY_REAL[3][5] + 1.1;
    RETAINTEST_AUTO_STRUCTUREARRAYARRAY.ARRAYARRAY_REAL[3][6] := RETAINTEST_AUTO_STRUCTUREARRAYARRAY.ARRAYARRAY_REAL[3][6] + 1.1;
    RETAINTEST_AUTO_STRUCTUREARRAYARRAY.ARRAYARRAY_REAL[3][7] := RETAINTEST_AUTO_STRUCTUREARRAYARRAY.ARRAYARRAY_REAL[3][7] + 1.1;
    RETAINTEST_AUTO_STRUCTUREARRAYARRAY.ARRAYARRAY_REAL[3][8] := RETAINTEST_AUTO_STRUCTUREARRAYARRAY.ARRAYARRAY_REAL[3][8] + 1.1;
    RETAINTEST_AUTO_STRUCTUREARRAYARRAY.ARRAYARRAY_REAL[3][9] := RETAINTEST_AUTO_STRUCTUREARRAYARRAY.ARRAYARRAY_REAL[3][9] + 1.1;

    RETAINTEST_AUTO_STRUCTUREARRAYARRAY.ARRAYARRAY_REAL[4][0] := RETAINTEST_AUTO_STRUCTUREARRAYARRAY.ARRAYARRAY_REAL[4][0] + 1.1;
    RETAINTEST_AUTO_STRUCTUREARRAYARRAY.ARRAYARRAY_REAL[4][1] := RETAINTEST_AUTO_STRUCTUREARRAYARRAY.ARRAYARRAY_REAL[4][1] + 1.1;
    RETAINTEST_AUTO_STRUCTUREARRAYARRAY.ARRAYARRAY_REAL[4][2] := RETAINTEST_AUTO_STRUCTUREARRAYARRAY.ARRAYARRAY_REAL[4][2] + 1.1;
    RETAINTEST_AUTO_STRUCTUREARRAYARRAY.ARRAYARRAY_REAL[4][3] := RETAINTEST_AUTO_STRUCTUREARRAYARRAY.ARRAYARRAY_REAL[4][3] + 1.1;
    RETAINTEST_AUTO_STRUCTUREARRAYARRAY.ARRAYARRAY_REAL[4][4] := RETAINTEST_AUTO_STRUCTUREARRAYARRAY.ARRAYARRAY_REAL[4][4] + 1.1;
    RETAINTEST_AUTO_STRUCTUREARRAYARRAY.ARRAYARRAY_REAL[4][5] := RETAINTEST_AUTO_STRUCTUREARRAYARRAY.ARRAYARRAY_REAL[4][5] + 1.1;
    RETAINTEST_AUTO_STRUCTUREARRAYARRAY.ARRAYARRAY_REAL[4][6] := RETAINTEST_AUTO_STRUCTUREARRAYARRAY.ARRAYARRAY_REAL[4][6] + 1.1;
    RETAINTEST_AUTO_STRUCTUREARRAYARRAY.ARRAYARRAY_REAL[4][7] := RETAINTEST_AUTO_STRUCTUREARRAYARRAY.ARRAYARRAY_REAL[4][7] + 1.1;
    RETAINTEST_AUTO_STRUCTUREARRAYARRAY.ARRAYARRAY_REAL[4][8] := RETAINTEST_AUTO_STRUCTUREARRAYARRAY.ARRAYARRAY_REAL[4][8] + 1.1;
    RETAINTEST_AUTO_STRUCTUREARRAYARRAY.ARRAYARRAY_REAL[4][9] := RETAINTEST_AUTO_STRUCTUREARRAYARRAY.ARRAYARRAY_REAL[4][9] + 1.1;

    RETAINTEST_AUTO_STRUCTUREARRAYARRAY.ARRAYARRAY_REAL[5][0] := RETAINTEST_AUTO_STRUCTUREARRAYARRAY.ARRAYARRAY_REAL[5][0] + 1.1;
    RETAINTEST_AUTO_STRUCTUREARRAYARRAY.ARRAYARRAY_REAL[5][1] := RETAINTEST_AUTO_STRUCTUREARRAYARRAY.ARRAYARRAY_REAL[5][1] + 1.1;
    RETAINTEST_AUTO_STRUCTUREARRAYARRAY.ARRAYARRAY_REAL[5][2] := RETAINTEST_AUTO_STRUCTUREARRAYARRAY.ARRAYARRAY_REAL[5][2] + 1.1;
    RETAINTEST_AUTO_STRUCTUREARRAYARRAY.ARRAYARRAY_REAL[5][3] := RETAINTEST_AUTO_STRUCTUREARRAYARRAY.ARRAYARRAY_REAL[5][3] + 1.1;
    RETAINTEST_AUTO_STRUCTUREARRAYARRAY.ARRAYARRAY_REAL[5][4] := RETAINTEST_AUTO_STRUCTUREARRAYARRAY.ARRAYARRAY_REAL[5][4] + 1.1;
    RETAINTEST_AUTO_STRUCTUREARRAYARRAY.ARRAYARRAY_REAL[5][5] := RETAINTEST_AUTO_STRUCTUREARRAYARRAY.ARRAYARRAY_REAL[5][5] + 1.1;
    RETAINTEST_AUTO_STRUCTUREARRAYARRAY.ARRAYARRAY_REAL[5][6] := RETAINTEST_AUTO_STRUCTUREARRAYARRAY.ARRAYARRAY_REAL[5][6] + 1.1;
    RETAINTEST_AUTO_STRUCTUREARRAYARRAY.ARRAYARRAY_REAL[5][7] := RETAINTEST_AUTO_STRUCTUREARRAYARRAY.ARRAYARRAY_REAL[5][7] + 1.1;
    RETAINTEST_AUTO_STRUCTUREARRAYARRAY.ARRAYARRAY_REAL[5][8] := RETAINTEST_AUTO_STRUCTUREARRAYARRAY.ARRAYARRAY_REAL[5][8] + 1.1;
    RETAINTEST_AUTO_STRUCTUREARRAYARRAY.ARRAYARRAY_REAL[5][9] := RETAINTEST_AUTO_STRUCTUREARRAYARRAY.ARRAYARRAY_REAL[5][9] + 1.1;

    RETAINTEST_AUTO_STRUCTUREARRAYARRAY.ARRAYARRAY_REAL[6][0] := RETAINTEST_AUTO_STRUCTUREARRAYARRAY.ARRAYARRAY_REAL[6][0] + 1.1;
    RETAINTEST_AUTO_STRUCTUREARRAYARRAY.ARRAYARRAY_REAL[6][1] := RETAINTEST_AUTO_STRUCTUREARRAYARRAY.ARRAYARRAY_REAL[6][1] + 1.1;
    RETAINTEST_AUTO_STRUCTUREARRAYARRAY.ARRAYARRAY_REAL[6][2] := RETAINTEST_AUTO_STRUCTUREARRAYARRAY.ARRAYARRAY_REAL[6][2] + 1.1;
    RETAINTEST_AUTO_STRUCTUREARRAYARRAY.ARRAYARRAY_REAL[6][3] := RETAINTEST_AUTO_STRUCTUREARRAYARRAY.ARRAYARRAY_REAL[6][3] + 1.1;
    RETAINTEST_AUTO_STRUCTUREARRAYARRAY.ARRAYARRAY_REAL[6][4] := RETAINTEST_AUTO_STRUCTUREARRAYARRAY.ARRAYARRAY_REAL[6][4] + 1.1;
    RETAINTEST_AUTO_STRUCTUREARRAYARRAY.ARRAYARRAY_REAL[6][5] := RETAINTEST_AUTO_STRUCTUREARRAYARRAY.ARRAYARRAY_REAL[6][5] + 1.1;
    RETAINTEST_AUTO_STRUCTUREARRAYARRAY.ARRAYARRAY_REAL[6][6] := RETAINTEST_AUTO_STRUCTUREARRAYARRAY.ARRAYARRAY_REAL[6][6] + 1.1;
    RETAINTEST_AUTO_STRUCTUREARRAYARRAY.ARRAYARRAY_REAL[6][7] := RETAINTEST_AUTO_STRUCTUREARRAYARRAY.ARRAYARRAY_REAL[6][7] + 1.1;
    RETAINTEST_AUTO_STRUCTUREARRAYARRAY.ARRAYARRAY_REAL[6][8] := RETAINTEST_AUTO_STRUCTUREARRAYARRAY.ARRAYARRAY_REAL[6][8] + 1.1;
    RETAINTEST_AUTO_STRUCTUREARRAYARRAY.ARRAYARRAY_REAL[6][9] := RETAINTEST_AUTO_STRUCTUREARRAYARRAY.ARRAYARRAY_REAL[6][9] + 1.1;

    RETAINTEST_AUTO_STRUCTUREARRAYARRAY.ARRAYARRAY_REAL[7][0] := RETAINTEST_AUTO_STRUCTUREARRAYARRAY.ARRAYARRAY_REAL[6][0];
    RETAINTEST_AUTO_STRUCTUREARRAYARRAY.ARRAYARRAY_REAL[7][1] := RETAINTEST_AUTO_STRUCTUREARRAYARRAY.ARRAYARRAY_REAL[6][1];
    RETAINTEST_AUTO_STRUCTUREARRAYARRAY.ARRAYARRAY_REAL[7][2] := RETAINTEST_AUTO_STRUCTUREARRAYARRAY.ARRAYARRAY_REAL[6][2];
    RETAINTEST_AUTO_STRUCTUREARRAYARRAY.ARRAYARRAY_REAL[7][3] := RETAINTEST_AUTO_STRUCTUREARRAYARRAY.ARRAYARRAY_REAL[6][3];
    RETAINTEST_AUTO_STRUCTUREARRAYARRAY.ARRAYARRAY_REAL[7][4] := RETAINTEST_AUTO_STRUCTUREARRAYARRAY.ARRAYARRAY_REAL[6][4];
    RETAINTEST_AUTO_STRUCTUREARRAYARRAY.ARRAYARRAY_REAL[7][5] := RETAINTEST_AUTO_STRUCTUREARRAYARRAY.ARRAYARRAY_REAL[6][5];
    RETAINTEST_AUTO_STRUCTUREARRAYARRAY.ARRAYARRAY_REAL[7][6] := RETAINTEST_AUTO_STRUCTUREARRAYARRAY.ARRAYARRAY_REAL[6][6];
    RETAINTEST_AUTO_STRUCTUREARRAYARRAY.ARRAYARRAY_REAL[7][7] := RETAINTEST_AUTO_STRUCTUREARRAYARRAY.ARRAYARRAY_REAL[6][7];
    RETAINTEST_AUTO_STRUCTUREARRAYARRAY.ARRAYARRAY_REAL[7][8] := RETAINTEST_AUTO_STRUCTUREARRAYARRAY.ARRAYARRAY_REAL[6][8];
    RETAINTEST_AUTO_STRUCTUREARRAYARRAY.ARRAYARRAY_REAL[7][9] := RETAINTEST_AUTO_STRUCTUREARRAYARRAY.ARRAYARRAY_REAL[6][9];

    RETAINTEST_AUTO_STRUCTUREARRAYARRAY.ARRAYARRAY_SINT[0][0] := RETAINTEST_AUTO_STRUCTUREARRAYARRAY.ARRAYARRAY_SINT[0][0] + 1;
    RETAINTEST_AUTO_STRUCTUREARRAYARRAY.ARRAYARRAY_SINT[0][1] := RETAINTEST_AUTO_STRUCTUREARRAYARRAY.ARRAYARRAY_SINT[0][1] + 1;
    RETAINTEST_AUTO_STRUCTUREARRAYARRAY.ARRAYARRAY_SINT[0][2] := RETAINTEST_AUTO_STRUCTUREARRAYARRAY.ARRAYARRAY_SINT[0][2] + 1;
    RETAINTEST_AUTO_STRUCTUREARRAYARRAY.ARRAYARRAY_SINT[0][3] := RETAINTEST_AUTO_STRUCTUREARRAYARRAY.ARRAYARRAY_SINT[0][3] + 1;
    RETAINTEST_AUTO_STRUCTUREARRAYARRAY.ARRAYARRAY_SINT[0][4] := RETAINTEST_AUTO_STRUCTUREARRAYARRAY.ARRAYARRAY_SINT[0][4] + 1;
    RETAINTEST_AUTO_STRUCTUREARRAYARRAY.ARRAYARRAY_SINT[0][5] := RETAINTEST_AUTO_STRUCTUREARRAYARRAY.ARRAYARRAY_SINT[0][5] + 1;
    RETAINTEST_AUTO_STRUCTUREARRAYARRAY.ARRAYARRAY_SINT[0][6] := RETAINTEST_AUTO_STRUCTUREARRAYARRAY.ARRAYARRAY_SINT[0][6] + 1;
    RETAINTEST_AUTO_STRUCTUREARRAYARRAY.ARRAYARRAY_SINT[0][7] := RETAINTEST_AUTO_STRUCTUREARRAYARRAY.ARRAYARRAY_SINT[0][7] + 1;
    RETAINTEST_AUTO_STRUCTUREARRAYARRAY.ARRAYARRAY_SINT[0][8] := RETAINTEST_AUTO_STRUCTUREARRAYARRAY.ARRAYARRAY_SINT[0][6];
    RETAINTEST_AUTO_STRUCTUREARRAYARRAY.ARRAYARRAY_SINT[0][9] := RETAINTEST_AUTO_STRUCTUREARRAYARRAY.ARRAYARRAY_SINT[0][7];

    RETAINTEST_AUTO_STRUCTUREARRAYARRAY.ARRAYARRAY_SINT[1][0] := RETAINTEST_AUTO_STRUCTUREARRAYARRAY.ARRAYARRAY_SINT[1][0] + 1;
    RETAINTEST_AUTO_STRUCTUREARRAYARRAY.ARRAYARRAY_SINT[1][1] := RETAINTEST_AUTO_STRUCTUREARRAYARRAY.ARRAYARRAY_SINT[1][1] + 1;
    RETAINTEST_AUTO_STRUCTUREARRAYARRAY.ARRAYARRAY_SINT[1][2] := RETAINTEST_AUTO_STRUCTUREARRAYARRAY.ARRAYARRAY_SINT[1][2] + 1;
    RETAINTEST_AUTO_STRUCTUREARRAYARRAY.ARRAYARRAY_SINT[1][3] := RETAINTEST_AUTO_STRUCTUREARRAYARRAY.ARRAYARRAY_SINT[1][3] + 1;
    RETAINTEST_AUTO_STRUCTUREARRAYARRAY.ARRAYARRAY_SINT[1][4] := RETAINTEST_AUTO_STRUCTUREARRAYARRAY.ARRAYARRAY_SINT[1][4] + 1;
    RETAINTEST_AUTO_STRUCTUREARRAYARRAY.ARRAYARRAY_SINT[1][5] := RETAINTEST_AUTO_STRUCTUREARRAYARRAY.ARRAYARRAY_SINT[1][5] + 1;
    RETAINTEST_AUTO_STRUCTUREARRAYARRAY.ARRAYARRAY_SINT[1][6] := RETAINTEST_AUTO_STRUCTUREARRAYARRAY.ARRAYARRAY_SINT[1][6] + 1;
    RETAINTEST_AUTO_STRUCTUREARRAYARRAY.ARRAYARRAY_SINT[1][7] := RETAINTEST_AUTO_STRUCTUREARRAYARRAY.ARRAYARRAY_SINT[1][7] + 1;
    RETAINTEST_AUTO_STRUCTUREARRAYARRAY.ARRAYARRAY_SINT[1][8] := RETAINTEST_AUTO_STRUCTUREARRAYARRAY.ARRAYARRAY_SINT[1][6];
    RETAINTEST_AUTO_STRUCTUREARRAYARRAY.ARRAYARRAY_SINT[1][9] := RETAINTEST_AUTO_STRUCTUREARRAYARRAY.ARRAYARRAY_SINT[1][7];

    RETAINTEST_AUTO_STRUCTUREARRAYARRAY.ARRAYARRAY_SINT[2][0] := RETAINTEST_AUTO_STRUCTUREARRAYARRAY.ARRAYARRAY_SINT[2][0] + 1;
    RETAINTEST_AUTO_STRUCTUREARRAYARRAY.ARRAYARRAY_SINT[2][1] := RETAINTEST_AUTO_STRUCTUREARRAYARRAY.ARRAYARRAY_SINT[2][1] + 1;
    RETAINTEST_AUTO_STRUCTUREARRAYARRAY.ARRAYARRAY_SINT[2][2] := RETAINTEST_AUTO_STRUCTUREARRAYARRAY.ARRAYARRAY_SINT[2][2] + 1;
    RETAINTEST_AUTO_STRUCTUREARRAYARRAY.ARRAYARRAY_SINT[2][3] := RETAINTEST_AUTO_STRUCTUREARRAYARRAY.ARRAYARRAY_SINT[2][3] + 1;
    RETAINTEST_AUTO_STRUCTUREARRAYARRAY.ARRAYARRAY_SINT[2][4] := RETAINTEST_AUTO_STRUCTUREARRAYARRAY.ARRAYARRAY_SINT[2][4] + 1;
    RETAINTEST_AUTO_STRUCTUREARRAYARRAY.ARRAYARRAY_SINT[2][5] := RETAINTEST_AUTO_STRUCTUREARRAYARRAY.ARRAYARRAY_SINT[2][5] + 1;
    RETAINTEST_AUTO_STRUCTUREARRAYARRAY.ARRAYARRAY_SINT[2][6] := RETAINTEST_AUTO_STRUCTUREARRAYARRAY.ARRAYARRAY_SINT[2][6] + 1;
    RETAINTEST_AUTO_STRUCTUREARRAYARRAY.ARRAYARRAY_SINT[2][7] := RETAINTEST_AUTO_STRUCTUREARRAYARRAY.ARRAYARRAY_SINT[2][7] + 1;
    RETAINTEST_AUTO_STRUCTUREARRAYARRAY.ARRAYARRAY_SINT[2][8] := RETAINTEST_AUTO_STRUCTUREARRAYARRAY.ARRAYARRAY_SINT[2][8] + 1;
    RETAINTEST_AUTO_STRUCTUREARRAYARRAY.ARRAYARRAY_SINT[2][9] := RETAINTEST_AUTO_STRUCTUREARRAYARRAY.ARRAYARRAY_SINT[2][9] + 1;

    RETAINTEST_AUTO_STRUCTUREARRAYARRAY.ARRAYARRAY_SINT[3][0] := RETAINTEST_AUTO_STRUCTUREARRAYARRAY.ARRAYARRAY_SINT[3][0] + 1;
    RETAINTEST_AUTO_STRUCTUREARRAYARRAY.ARRAYARRAY_SINT[3][1] := RETAINTEST_AUTO_STRUCTUREARRAYARRAY.ARRAYARRAY_SINT[3][1] + 1;
    RETAINTEST_AUTO_STRUCTUREARRAYARRAY.ARRAYARRAY_SINT[3][2] := RETAINTEST_AUTO_STRUCTUREARRAYARRAY.ARRAYARRAY_SINT[3][2] + 1;
    RETAINTEST_AUTO_STRUCTUREARRAYARRAY.ARRAYARRAY_SINT[3][3] := RETAINTEST_AUTO_STRUCTUREARRAYARRAY.ARRAYARRAY_SINT[3][3] + 1;
    RETAINTEST_AUTO_STRUCTUREARRAYARRAY.ARRAYARRAY_SINT[3][4] := RETAINTEST_AUTO_STRUCTUREARRAYARRAY.ARRAYARRAY_SINT[3][4] + 1;
    RETAINTEST_AUTO_STRUCTUREARRAYARRAY.ARRAYARRAY_SINT[3][5] := RETAINTEST_AUTO_STRUCTUREARRAYARRAY.ARRAYARRAY_SINT[3][5] + 1;
    RETAINTEST_AUTO_STRUCTUREARRAYARRAY.ARRAYARRAY_SINT[3][6] := RETAINTEST_AUTO_STRUCTUREARRAYARRAY.ARRAYARRAY_SINT[3][6] + 1;
    RETAINTEST_AUTO_STRUCTUREARRAYARRAY.ARRAYARRAY_SINT[3][7] := RETAINTEST_AUTO_STRUCTUREARRAYARRAY.ARRAYARRAY_SINT[3][7] + 1;
    RETAINTEST_AUTO_STRUCTUREARRAYARRAY.ARRAYARRAY_SINT[3][8] := RETAINTEST_AUTO_STRUCTUREARRAYARRAY.ARRAYARRAY_SINT[3][8] + 1;
    RETAINTEST_AUTO_STRUCTUREARRAYARRAY.ARRAYARRAY_SINT[3][9] := RETAINTEST_AUTO_STRUCTUREARRAYARRAY.ARRAYARRAY_SINT[3][9] + 1;

    RETAINTEST_AUTO_STRUCTUREARRAYARRAY.ARRAYARRAY_SINT[4][0] := RETAINTEST_AUTO_STRUCTUREARRAYARRAY.ARRAYARRAY_SINT[4][0] + 1;
    RETAINTEST_AUTO_STRUCTUREARRAYARRAY.ARRAYARRAY_SINT[4][1] := RETAINTEST_AUTO_STRUCTUREARRAYARRAY.ARRAYARRAY_SINT[4][1] + 1;
    RETAINTEST_AUTO_STRUCTUREARRAYARRAY.ARRAYARRAY_SINT[4][2] := RETAINTEST_AUTO_STRUCTUREARRAYARRAY.ARRAYARRAY_SINT[4][2] + 1;
    RETAINTEST_AUTO_STRUCTUREARRAYARRAY.ARRAYARRAY_SINT[4][3] := RETAINTEST_AUTO_STRUCTUREARRAYARRAY.ARRAYARRAY_SINT[4][3] + 1;
    RETAINTEST_AUTO_STRUCTUREARRAYARRAY.ARRAYARRAY_SINT[4][4] := RETAINTEST_AUTO_STRUCTUREARRAYARRAY.ARRAYARRAY_SINT[4][4] + 1;
    RETAINTEST_AUTO_STRUCTUREARRAYARRAY.ARRAYARRAY_SINT[4][5] := RETAINTEST_AUTO_STRUCTUREARRAYARRAY.ARRAYARRAY_SINT[4][5] + 1;
    RETAINTEST_AUTO_STRUCTUREARRAYARRAY.ARRAYARRAY_SINT[4][6] := RETAINTEST_AUTO_STRUCTUREARRAYARRAY.ARRAYARRAY_SINT[4][6] + 1;
    RETAINTEST_AUTO_STRUCTUREARRAYARRAY.ARRAYARRAY_SINT[4][7] := RETAINTEST_AUTO_STRUCTUREARRAYARRAY.ARRAYARRAY_SINT[4][7] + 1;
    RETAINTEST_AUTO_STRUCTUREARRAYARRAY.ARRAYARRAY_SINT[4][8] := RETAINTEST_AUTO_STRUCTUREARRAYARRAY.ARRAYARRAY_SINT[4][8] + 1;
    RETAINTEST_AUTO_STRUCTUREARRAYARRAY.ARRAYARRAY_SINT[4][9] := RETAINTEST_AUTO_STRUCTUREARRAYARRAY.ARRAYARRAY_SINT[4][9] + 1;

    RETAINTEST_AUTO_STRUCTUREARRAYARRAY.ARRAYARRAY_SINT[5][0] := RETAINTEST_AUTO_STRUCTUREARRAYARRAY.ARRAYARRAY_SINT[5][0] + 1;
    RETAINTEST_AUTO_STRUCTUREARRAYARRAY.ARRAYARRAY_SINT[5][1] := RETAINTEST_AUTO_STRUCTUREARRAYARRAY.ARRAYARRAY_SINT[5][1] + 1;
    RETAINTEST_AUTO_STRUCTUREARRAYARRAY.ARRAYARRAY_SINT[5][2] := RETAINTEST_AUTO_STRUCTUREARRAYARRAY.ARRAYARRAY_SINT[5][2] + 1;
    RETAINTEST_AUTO_STRUCTUREARRAYARRAY.ARRAYARRAY_SINT[5][3] := RETAINTEST_AUTO_STRUCTUREARRAYARRAY.ARRAYARRAY_SINT[5][3] + 1;
    RETAINTEST_AUTO_STRUCTUREARRAYARRAY.ARRAYARRAY_SINT[5][4] := RETAINTEST_AUTO_STRUCTUREARRAYARRAY.ARRAYARRAY_SINT[5][4] + 1;
    RETAINTEST_AUTO_STRUCTUREARRAYARRAY.ARRAYARRAY_SINT[5][5] := RETAINTEST_AUTO_STRUCTUREARRAYARRAY.ARRAYARRAY_SINT[5][5] + 1;
    RETAINTEST_AUTO_STRUCTUREARRAYARRAY.ARRAYARRAY_SINT[5][6] := RETAINTEST_AUTO_STRUCTUREARRAYARRAY.ARRAYARRAY_SINT[5][6] + 1;
    RETAINTEST_AUTO_STRUCTUREARRAYARRAY.ARRAYARRAY_SINT[5][7] := RETAINTEST_AUTO_STRUCTUREARRAYARRAY.ARRAYARRAY_SINT[5][7] + 1;
    RETAINTEST_AUTO_STRUCTUREARRAYARRAY.ARRAYARRAY_SINT[5][8] := RETAINTEST_AUTO_STRUCTUREARRAYARRAY.ARRAYARRAY_SINT[5][8] + 1;
    RETAINTEST_AUTO_STRUCTUREARRAYARRAY.ARRAYARRAY_SINT[5][9] := RETAINTEST_AUTO_STRUCTUREARRAYARRAY.ARRAYARRAY_SINT[5][9] + 1;

    RETAINTEST_AUTO_STRUCTUREARRAYARRAY.ARRAYARRAY_SINT[6][0] := RETAINTEST_AUTO_STRUCTUREARRAYARRAY.ARRAYARRAY_SINT[6][0] + 1;
    RETAINTEST_AUTO_STRUCTUREARRAYARRAY.ARRAYARRAY_SINT[6][1] := RETAINTEST_AUTO_STRUCTUREARRAYARRAY.ARRAYARRAY_SINT[6][1] + 1;
    RETAINTEST_AUTO_STRUCTUREARRAYARRAY.ARRAYARRAY_SINT[6][2] := RETAINTEST_AUTO_STRUCTUREARRAYARRAY.ARRAYARRAY_SINT[6][2] + 1;
    RETAINTEST_AUTO_STRUCTUREARRAYARRAY.ARRAYARRAY_SINT[6][3] := RETAINTEST_AUTO_STRUCTUREARRAYARRAY.ARRAYARRAY_SINT[6][3] + 1;
    RETAINTEST_AUTO_STRUCTUREARRAYARRAY.ARRAYARRAY_SINT[6][4] := RETAINTEST_AUTO_STRUCTUREARRAYARRAY.ARRAYARRAY_SINT[6][4] + 1;
    RETAINTEST_AUTO_STRUCTUREARRAYARRAY.ARRAYARRAY_SINT[6][5] := RETAINTEST_AUTO_STRUCTUREARRAYARRAY.ARRAYARRAY_SINT[6][5] + 1;
    RETAINTEST_AUTO_STRUCTUREARRAYARRAY.ARRAYARRAY_SINT[6][6] := RETAINTEST_AUTO_STRUCTUREARRAYARRAY.ARRAYARRAY_SINT[6][6] + 1;
    RETAINTEST_AUTO_STRUCTUREARRAYARRAY.ARRAYARRAY_SINT[6][7] := RETAINTEST_AUTO_STRUCTUREARRAYARRAY.ARRAYARRAY_SINT[6][7] + 1;
    RETAINTEST_AUTO_STRUCTUREARRAYARRAY.ARRAYARRAY_SINT[6][8] := RETAINTEST_AUTO_STRUCTUREARRAYARRAY.ARRAYARRAY_SINT[6][8] + 1;
    RETAINTEST_AUTO_STRUCTUREARRAYARRAY.ARRAYARRAY_SINT[6][9] := RETAINTEST_AUTO_STRUCTUREARRAYARRAY.ARRAYARRAY_SINT[6][9] + 1;

    RETAINTEST_AUTO_STRUCTUREARRAYARRAY.ARRAYARRAY_SINT[7][0] := RETAINTEST_AUTO_STRUCTUREARRAYARRAY.ARRAYARRAY_SINT[6][0];
    RETAINTEST_AUTO_STRUCTUREARRAYARRAY.ARRAYARRAY_SINT[7][1] := RETAINTEST_AUTO_STRUCTUREARRAYARRAY.ARRAYARRAY_SINT[6][1];
    RETAINTEST_AUTO_STRUCTUREARRAYARRAY.ARRAYARRAY_SINT[7][2] := RETAINTEST_AUTO_STRUCTUREARRAYARRAY.ARRAYARRAY_SINT[6][2];
    RETAINTEST_AUTO_STRUCTUREARRAYARRAY.ARRAYARRAY_SINT[7][3] := RETAINTEST_AUTO_STRUCTUREARRAYARRAY.ARRAYARRAY_SINT[6][3];
    RETAINTEST_AUTO_STRUCTUREARRAYARRAY.ARRAYARRAY_SINT[7][4] := RETAINTEST_AUTO_STRUCTUREARRAYARRAY.ARRAYARRAY_SINT[6][4];
    RETAINTEST_AUTO_STRUCTUREARRAYARRAY.ARRAYARRAY_SINT[7][5] := RETAINTEST_AUTO_STRUCTUREARRAYARRAY.ARRAYARRAY_SINT[6][5];
    RETAINTEST_AUTO_STRUCTUREARRAYARRAY.ARRAYARRAY_SINT[7][6] := RETAINTEST_AUTO_STRUCTUREARRAYARRAY.ARRAYARRAY_SINT[6][6];
    RETAINTEST_AUTO_STRUCTUREARRAYARRAY.ARRAYARRAY_SINT[7][7] := RETAINTEST_AUTO_STRUCTUREARRAYARRAY.ARRAYARRAY_SINT[6][7];
    RETAINTEST_AUTO_STRUCTUREARRAYARRAY.ARRAYARRAY_SINT[7][8] := RETAINTEST_AUTO_STRUCTUREARRAYARRAY.ARRAYARRAY_SINT[6][8];
    RETAINTEST_AUTO_STRUCTUREARRAYARRAY.ARRAYARRAY_SINT[7][9] := RETAINTEST_AUTO_STRUCTUREARRAYARRAY.ARRAYARRAY_SINT[6][9];

    RETAINTEST_AUTO_STRUCTUREARRAYARRAY.ARRAYARRAY_STRING[0][0] := ANY_TO_STRING(RETAINTEST_AUTO_ARRAYARRAY_DINT[0][0]) + ' ' + ANY_TO_STRING(RETAINTEST_AUTO_ARRAYARRAY_TIME[0][0]);
    RETAINTEST_AUTO_STRUCTUREARRAYARRAY.ARRAYARRAY_STRING[0][1] := ANY_TO_STRING(RETAINTEST_AUTO_ARRAYARRAY_DINT[0][1]) + ' ' + ANY_TO_STRING(RETAINTEST_AUTO_ARRAYARRAY_TIME[0][1]);
    RETAINTEST_AUTO_STRUCTUREARRAYARRAY.ARRAYARRAY_STRING[0][2] := ANY_TO_STRING(RETAINTEST_AUTO_ARRAYARRAY_DINT[0][2]) + ' ' + ANY_TO_STRING(RETAINTEST_AUTO_ARRAYARRAY_TIME[0][2]);
    RETAINTEST_AUTO_STRUCTUREARRAYARRAY.ARRAYARRAY_STRING[0][3] := ANY_TO_STRING(RETAINTEST_AUTO_ARRAYARRAY_DINT[0][3]) + ' ' + ANY_TO_STRING(RETAINTEST_AUTO_ARRAYARRAY_TIME[0][3]);
    RETAINTEST_AUTO_STRUCTUREARRAYARRAY.ARRAYARRAY_STRING[0][4] := ANY_TO_STRING(RETAINTEST_AUTO_ARRAYARRAY_DINT[0][4]) + ' ' + ANY_TO_STRING(RETAINTEST_AUTO_ARRAYARRAY_TIME[0][4]);
    RETAINTEST_AUTO_STRUCTUREARRAYARRAY.ARRAYARRAY_STRING[0][5] := ANY_TO_STRING(RETAINTEST_AUTO_ARRAYARRAY_DINT[0][5]) + ' ' + ANY_TO_STRING(RETAINTEST_AUTO_ARRAYARRAY_TIME[0][5]);
    RETAINTEST_AUTO_STRUCTUREARRAYARRAY.ARRAYARRAY_STRING[0][6] := ANY_TO_STRING(RETAINTEST_AUTO_ARRAYARRAY_DINT[0][6]) + ' ' + ANY_TO_STRING(RETAINTEST_AUTO_ARRAYARRAY_TIME[0][6]);
    RETAINTEST_AUTO_STRUCTUREARRAYARRAY.ARRAYARRAY_STRING[0][7] := ANY_TO_STRING(RETAINTEST_AUTO_ARRAYARRAY_DINT[0][7]) + ' ' + ANY_TO_STRING(RETAINTEST_AUTO_ARRAYARRAY_TIME[0][7]);
    RETAINTEST_AUTO_STRUCTUREARRAYARRAY.ARRAYARRAY_STRING[0][8] := RETAINTEST_AUTO_STRUCTUREARRAYARRAY.ARRAYARRAY_STRING[0][6];
    RETAINTEST_AUTO_STRUCTUREARRAYARRAY.ARRAYARRAY_STRING[0][9] := RETAINTEST_AUTO_STRUCTUREARRAYARRAY.ARRAYARRAY_STRING[0][7];

    RETAINTEST_AUTO_STRUCTUREARRAYARRAY.ARRAYARRAY_STRING[1][0] := ANY_TO_STRING(RETAINTEST_AUTO_ARRAYARRAY_DINT[1][0]) + ' ' + ANY_TO_STRING(RETAINTEST_AUTO_ARRAYARRAY_TIME[1][0]);
    RETAINTEST_AUTO_STRUCTUREARRAYARRAY.ARRAYARRAY_STRING[1][1] := ANY_TO_STRING(RETAINTEST_AUTO_ARRAYARRAY_DINT[1][1]) + ' ' + ANY_TO_STRING(RETAINTEST_AUTO_ARRAYARRAY_TIME[1][1]);
    RETAINTEST_AUTO_STRUCTUREARRAYARRAY.ARRAYARRAY_STRING[1][2] := ANY_TO_STRING(RETAINTEST_AUTO_ARRAYARRAY_DINT[1][2]) + ' ' + ANY_TO_STRING(RETAINTEST_AUTO_ARRAYARRAY_TIME[1][2]);
    RETAINTEST_AUTO_STRUCTUREARRAYARRAY.ARRAYARRAY_STRING[1][3] := ANY_TO_STRING(RETAINTEST_AUTO_ARRAYARRAY_DINT[1][3]) + ' ' + ANY_TO_STRING(RETAINTEST_AUTO_ARRAYARRAY_TIME[1][3]);
    RETAINTEST_AUTO_STRUCTUREARRAYARRAY.ARRAYARRAY_STRING[1][4] := ANY_TO_STRING(RETAINTEST_AUTO_ARRAYARRAY_DINT[1][4]) + ' ' + ANY_TO_STRING(RETAINTEST_AUTO_ARRAYARRAY_TIME[1][4]);
    RETAINTEST_AUTO_STRUCTUREARRAYARRAY.ARRAYARRAY_STRING[1][5] := ANY_TO_STRING(RETAINTEST_AUTO_ARRAYARRAY_DINT[1][5]) + ' ' + ANY_TO_STRING(RETAINTEST_AUTO_ARRAYARRAY_TIME[1][5]);
    RETAINTEST_AUTO_STRUCTUREARRAYARRAY.ARRAYARRAY_STRING[1][6] := ANY_TO_STRING(RETAINTEST_AUTO_ARRAYARRAY_DINT[1][6]) + ' ' + ANY_TO_STRING(RETAINTEST_AUTO_ARRAYARRAY_TIME[1][6]);
    RETAINTEST_AUTO_STRUCTUREARRAYARRAY.ARRAYARRAY_STRING[1][7] := ANY_TO_STRING(RETAINTEST_AUTO_ARRAYARRAY_DINT[1][7]) + ' ' + ANY_TO_STRING(RETAINTEST_AUTO_ARRAYARRAY_TIME[1][7]);
    RETAINTEST_AUTO_STRUCTUREARRAYARRAY.ARRAYARRAY_STRING[1][8] := RETAINTEST_AUTO_STRUCTUREARRAYARRAY.ARRAYARRAY_STRING[1][6];
    RETAINTEST_AUTO_STRUCTUREARRAYARRAY.ARRAYARRAY_STRING[1][9] := RETAINTEST_AUTO_STRUCTUREARRAYARRAY.ARRAYARRAY_STRING[1][7];

    RETAINTEST_AUTO_STRUCTUREARRAYARRAY.ARRAYARRAY_STRING[2][0] := ANY_TO_STRING(RETAINTEST_AUTO_ARRAYARRAY_DINT[2][0]) + ' ' + ANY_TO_STRING(RETAINTEST_AUTO_ARRAYARRAY_TIME[2][0]);
    RETAINTEST_AUTO_STRUCTUREARRAYARRAY.ARRAYARRAY_STRING[2][1] := ANY_TO_STRING(RETAINTEST_AUTO_ARRAYARRAY_DINT[2][1]) + ' ' + ANY_TO_STRING(RETAINTEST_AUTO_ARRAYARRAY_TIME[2][1]);
    RETAINTEST_AUTO_STRUCTUREARRAYARRAY.ARRAYARRAY_STRING[2][2] := ANY_TO_STRING(RETAINTEST_AUTO_ARRAYARRAY_DINT[2][2]) + ' ' + ANY_TO_STRING(RETAINTEST_AUTO_ARRAYARRAY_TIME[2][2]);
    RETAINTEST_AUTO_STRUCTUREARRAYARRAY.ARRAYARRAY_STRING[2][3] := ANY_TO_STRING(RETAINTEST_AUTO_ARRAYARRAY_DINT[2][3]) + ' ' + ANY_TO_STRING(RETAINTEST_AUTO_ARRAYARRAY_TIME[2][3]);
    RETAINTEST_AUTO_STRUCTUREARRAYARRAY.ARRAYARRAY_STRING[2][4] := ANY_TO_STRING(RETAINTEST_AUTO_ARRAYARRAY_DINT[2][4]) + ' ' + ANY_TO_STRING(RETAINTEST_AUTO_ARRAYARRAY_TIME[2][4]);
    RETAINTEST_AUTO_STRUCTUREARRAYARRAY.ARRAYARRAY_STRING[2][5] := ANY_TO_STRING(RETAINTEST_AUTO_ARRAYARRAY_DINT[2][5]) + ' ' + ANY_TO_STRING(RETAINTEST_AUTO_ARRAYARRAY_TIME[2][5]);
    RETAINTEST_AUTO_STRUCTUREARRAYARRAY.ARRAYARRAY_STRING[2][6] := ANY_TO_STRING(RETAINTEST_AUTO_ARRAYARRAY_DINT[2][6]) + ' ' + ANY_TO_STRING(RETAINTEST_AUTO_ARRAYARRAY_TIME[2][6]);
    RETAINTEST_AUTO_STRUCTUREARRAYARRAY.ARRAYARRAY_STRING[2][7] := ANY_TO_STRING(RETAINTEST_AUTO_ARRAYARRAY_DINT[2][7]) + ' ' + ANY_TO_STRING(RETAINTEST_AUTO_ARRAYARRAY_TIME[2][7]);
    RETAINTEST_AUTO_STRUCTUREARRAYARRAY.ARRAYARRAY_STRING[2][8] := ANY_TO_STRING(RETAINTEST_AUTO_ARRAYARRAY_DINT[2][8]) + ' ' + ANY_TO_STRING(RETAINTEST_AUTO_ARRAYARRAY_TIME[2][8]);
    RETAINTEST_AUTO_STRUCTUREARRAYARRAY.ARRAYARRAY_STRING[2][9] := ANY_TO_STRING(RETAINTEST_AUTO_ARRAYARRAY_DINT[2][9]) + ' ' + ANY_TO_STRING(RETAINTEST_AUTO_ARRAYARRAY_TIME[2][9]);

    RETAINTEST_AUTO_STRUCTUREARRAYARRAY.ARRAYARRAY_STRING[3][0] := ANY_TO_STRING(RETAINTEST_AUTO_ARRAYARRAY_DINT[3][0]) + ' ' + ANY_TO_STRING(RETAINTEST_AUTO_ARRAYARRAY_TIME[3][0]);
    RETAINTEST_AUTO_STRUCTUREARRAYARRAY.ARRAYARRAY_STRING[3][1] := ANY_TO_STRING(RETAINTEST_AUTO_ARRAYARRAY_DINT[3][1]) + ' ' + ANY_TO_STRING(RETAINTEST_AUTO_ARRAYARRAY_TIME[3][1]);
    RETAINTEST_AUTO_STRUCTUREARRAYARRAY.ARRAYARRAY_STRING[3][2] := ANY_TO_STRING(RETAINTEST_AUTO_ARRAYARRAY_DINT[3][2]) + ' ' + ANY_TO_STRING(RETAINTEST_AUTO_ARRAYARRAY_TIME[3][2]);
    RETAINTEST_AUTO_STRUCTUREARRAYARRAY.ARRAYARRAY_STRING[3][3] := ANY_TO_STRING(RETAINTEST_AUTO_ARRAYARRAY_DINT[3][3]) + ' ' + ANY_TO_STRING(RETAINTEST_AUTO_ARRAYARRAY_TIME[3][3]);
    RETAINTEST_AUTO_STRUCTUREARRAYARRAY.ARRAYARRAY_STRING[3][4] := ANY_TO_STRING(RETAINTEST_AUTO_ARRAYARRAY_DINT[3][4]) + ' ' + ANY_TO_STRING(RETAINTEST_AUTO_ARRAYARRAY_TIME[3][4]);
    RETAINTEST_AUTO_STRUCTUREARRAYARRAY.ARRAYARRAY_STRING[3][5] := ANY_TO_STRING(RETAINTEST_AUTO_ARRAYARRAY_DINT[3][5]) + ' ' + ANY_TO_STRING(RETAINTEST_AUTO_ARRAYARRAY_TIME[3][5]);
    RETAINTEST_AUTO_STRUCTUREARRAYARRAY.ARRAYARRAY_STRING[3][6] := ANY_TO_STRING(RETAINTEST_AUTO_ARRAYARRAY_DINT[3][6]) + ' ' + ANY_TO_STRING(RETAINTEST_AUTO_ARRAYARRAY_TIME[3][6]);
    RETAINTEST_AUTO_STRUCTUREARRAYARRAY.ARRAYARRAY_STRING[3][7] := ANY_TO_STRING(RETAINTEST_AUTO_ARRAYARRAY_DINT[3][7]) + ' ' + ANY_TO_STRING(RETAINTEST_AUTO_ARRAYARRAY_TIME[3][7]);
    RETAINTEST_AUTO_STRUCTUREARRAYARRAY.ARRAYARRAY_STRING[3][8] := ANY_TO_STRING(RETAINTEST_AUTO_ARRAYARRAY_DINT[3][8]) + ' ' + ANY_TO_STRING(RETAINTEST_AUTO_ARRAYARRAY_TIME[3][8]);
    RETAINTEST_AUTO_STRUCTUREARRAYARRAY.ARRAYARRAY_STRING[3][9] := ANY_TO_STRING(RETAINTEST_AUTO_ARRAYARRAY_DINT[3][9]) + ' ' + ANY_TO_STRING(RETAINTEST_AUTO_ARRAYARRAY_TIME[3][9]);

    RETAINTEST_AUTO_STRUCTUREARRAYARRAY.ARRAYARRAY_STRING[4][0] := ANY_TO_STRING(RETAINTEST_AUTO_ARRAYARRAY_DINT[4][0]) + ' ' + ANY_TO_STRING(RETAINTEST_AUTO_ARRAYARRAY_TIME[4][0]);
    RETAINTEST_AUTO_STRUCTUREARRAYARRAY.ARRAYARRAY_STRING[4][1] := ANY_TO_STRING(RETAINTEST_AUTO_ARRAYARRAY_DINT[4][1]) + ' ' + ANY_TO_STRING(RETAINTEST_AUTO_ARRAYARRAY_TIME[4][1]);
    RETAINTEST_AUTO_STRUCTUREARRAYARRAY.ARRAYARRAY_STRING[4][2] := ANY_TO_STRING(RETAINTEST_AUTO_ARRAYARRAY_DINT[4][2]) + ' ' + ANY_TO_STRING(RETAINTEST_AUTO_ARRAYARRAY_TIME[4][2]);
    RETAINTEST_AUTO_STRUCTUREARRAYARRAY.ARRAYARRAY_STRING[4][3] := ANY_TO_STRING(RETAINTEST_AUTO_ARRAYARRAY_DINT[4][3]) + ' ' + ANY_TO_STRING(RETAINTEST_AUTO_ARRAYARRAY_TIME[4][3]);
    RETAINTEST_AUTO_STRUCTUREARRAYARRAY.ARRAYARRAY_STRING[4][4] := ANY_TO_STRING(RETAINTEST_AUTO_ARRAYARRAY_DINT[4][4]) + ' ' + ANY_TO_STRING(RETAINTEST_AUTO_ARRAYARRAY_TIME[4][4]);
    RETAINTEST_AUTO_STRUCTUREARRAYARRAY.ARRAYARRAY_STRING[4][5] := ANY_TO_STRING(RETAINTEST_AUTO_ARRAYARRAY_DINT[4][5]) + ' ' + ANY_TO_STRING(RETAINTEST_AUTO_ARRAYARRAY_TIME[4][5]);
    RETAINTEST_AUTO_STRUCTUREARRAYARRAY.ARRAYARRAY_STRING[4][6] := ANY_TO_STRING(RETAINTEST_AUTO_ARRAYARRAY_DINT[4][6]) + ' ' + ANY_TO_STRING(RETAINTEST_AUTO_ARRAYARRAY_TIME[4][6]);
    RETAINTEST_AUTO_STRUCTUREARRAYARRAY.ARRAYARRAY_STRING[4][7] := ANY_TO_STRING(RETAINTEST_AUTO_ARRAYARRAY_DINT[4][7]) + ' ' + ANY_TO_STRING(RETAINTEST_AUTO_ARRAYARRAY_TIME[4][7]);
    RETAINTEST_AUTO_STRUCTUREARRAYARRAY.ARRAYARRAY_STRING[4][8] := ANY_TO_STRING(RETAINTEST_AUTO_ARRAYARRAY_DINT[4][8]) + ' ' + ANY_TO_STRING(RETAINTEST_AUTO_ARRAYARRAY_TIME[4][8]);
    RETAINTEST_AUTO_STRUCTUREARRAYARRAY.ARRAYARRAY_STRING[4][9] := ANY_TO_STRING(RETAINTEST_AUTO_ARRAYARRAY_DINT[4][9]) + ' ' + ANY_TO_STRING(RETAINTEST_AUTO_ARRAYARRAY_TIME[4][9]);

    RETAINTEST_AUTO_STRUCTUREARRAYARRAY.ARRAYARRAY_STRING[5][0] := ANY_TO_STRING(RETAINTEST_AUTO_ARRAYARRAY_DINT[5][0]) + ' ' + ANY_TO_STRING(RETAINTEST_AUTO_ARRAYARRAY_TIME[5][0]);
    RETAINTEST_AUTO_STRUCTUREARRAYARRAY.ARRAYARRAY_STRING[5][1] := ANY_TO_STRING(RETAINTEST_AUTO_ARRAYARRAY_DINT[5][1]) + ' ' + ANY_TO_STRING(RETAINTEST_AUTO_ARRAYARRAY_TIME[5][1]);
    RETAINTEST_AUTO_STRUCTUREARRAYARRAY.ARRAYARRAY_STRING[5][2] := ANY_TO_STRING(RETAINTEST_AUTO_ARRAYARRAY_DINT[5][2]) + ' ' + ANY_TO_STRING(RETAINTEST_AUTO_ARRAYARRAY_TIME[5][2]);
    RETAINTEST_AUTO_STRUCTUREARRAYARRAY.ARRAYARRAY_STRING[5][3] := ANY_TO_STRING(RETAINTEST_AUTO_ARRAYARRAY_DINT[5][3]) + ' ' + ANY_TO_STRING(RETAINTEST_AUTO_ARRAYARRAY_TIME[5][3]);
    RETAINTEST_AUTO_STRUCTUREARRAYARRAY.ARRAYARRAY_STRING[5][4] := ANY_TO_STRING(RETAINTEST_AUTO_ARRAYARRAY_DINT[5][4]) + ' ' + ANY_TO_STRING(RETAINTEST_AUTO_ARRAYARRAY_TIME[5][4]);
    RETAINTEST_AUTO_STRUCTUREARRAYARRAY.ARRAYARRAY_STRING[5][5] := ANY_TO_STRING(RETAINTEST_AUTO_ARRAYARRAY_DINT[5][5]) + ' ' + ANY_TO_STRING(RETAINTEST_AUTO_ARRAYARRAY_TIME[5][5]);
    RETAINTEST_AUTO_STRUCTUREARRAYARRAY.ARRAYARRAY_STRING[5][6] := ANY_TO_STRING(RETAINTEST_AUTO_ARRAYARRAY_DINT[5][6]) + ' ' + ANY_TO_STRING(RETAINTEST_AUTO_ARRAYARRAY_TIME[5][6]);
    RETAINTEST_AUTO_STRUCTUREARRAYARRAY.ARRAYARRAY_STRING[5][7] := ANY_TO_STRING(RETAINTEST_AUTO_ARRAYARRAY_DINT[5][7]) + ' ' + ANY_TO_STRING(RETAINTEST_AUTO_ARRAYARRAY_TIME[5][7]);
    RETAINTEST_AUTO_STRUCTUREARRAYARRAY.ARRAYARRAY_STRING[5][8] := ANY_TO_STRING(RETAINTEST_AUTO_ARRAYARRAY_DINT[5][8]) + ' ' + ANY_TO_STRING(RETAINTEST_AUTO_ARRAYARRAY_TIME[5][8]);
    RETAINTEST_AUTO_STRUCTUREARRAYARRAY.ARRAYARRAY_STRING[5][9] := ANY_TO_STRING(RETAINTEST_AUTO_ARRAYARRAY_DINT[5][9]) + ' ' + ANY_TO_STRING(RETAINTEST_AUTO_ARRAYARRAY_TIME[5][9]);

    RETAINTEST_AUTO_STRUCTUREARRAYARRAY.ARRAYARRAY_STRING[6][0] := ANY_TO_STRING(RETAINTEST_AUTO_ARRAYARRAY_DINT[6][0]) + ' ' + ANY_TO_STRING(RETAINTEST_AUTO_ARRAYARRAY_TIME[6][0]);
    RETAINTEST_AUTO_STRUCTUREARRAYARRAY.ARRAYARRAY_STRING[6][1] := ANY_TO_STRING(RETAINTEST_AUTO_ARRAYARRAY_DINT[6][1]) + ' ' + ANY_TO_STRING(RETAINTEST_AUTO_ARRAYARRAY_TIME[6][1]);
    RETAINTEST_AUTO_STRUCTUREARRAYARRAY.ARRAYARRAY_STRING[6][2] := ANY_TO_STRING(RETAINTEST_AUTO_ARRAYARRAY_DINT[6][2]) + ' ' + ANY_TO_STRING(RETAINTEST_AUTO_ARRAYARRAY_TIME[6][2]);
    RETAINTEST_AUTO_STRUCTUREARRAYARRAY.ARRAYARRAY_STRING[6][3] := ANY_TO_STRING(RETAINTEST_AUTO_ARRAYARRAY_DINT[6][3]) + ' ' + ANY_TO_STRING(RETAINTEST_AUTO_ARRAYARRAY_TIME[6][3]);
    RETAINTEST_AUTO_STRUCTUREARRAYARRAY.ARRAYARRAY_STRING[6][4] := ANY_TO_STRING(RETAINTEST_AUTO_ARRAYARRAY_DINT[6][4]) + ' ' + ANY_TO_STRING(RETAINTEST_AUTO_ARRAYARRAY_TIME[6][4]);
    RETAINTEST_AUTO_STRUCTUREARRAYARRAY.ARRAYARRAY_STRING[6][5] := ANY_TO_STRING(RETAINTEST_AUTO_ARRAYARRAY_DINT[6][5]) + ' ' + ANY_TO_STRING(RETAINTEST_AUTO_ARRAYARRAY_TIME[6][5]);
    RETAINTEST_AUTO_STRUCTUREARRAYARRAY.ARRAYARRAY_STRING[6][6] := ANY_TO_STRING(RETAINTEST_AUTO_ARRAYARRAY_DINT[6][6]) + ' ' + ANY_TO_STRING(RETAINTEST_AUTO_ARRAYARRAY_TIME[6][6]);
    RETAINTEST_AUTO_STRUCTUREARRAYARRAY.ARRAYARRAY_STRING[6][7] := ANY_TO_STRING(RETAINTEST_AUTO_ARRAYARRAY_DINT[6][7]) + ' ' + ANY_TO_STRING(RETAINTEST_AUTO_ARRAYARRAY_TIME[6][7]);
    RETAINTEST_AUTO_STRUCTUREARRAYARRAY.ARRAYARRAY_STRING[6][8] := ANY_TO_STRING(RETAINTEST_AUTO_ARRAYARRAY_DINT[6][8]) + ' ' + ANY_TO_STRING(RETAINTEST_AUTO_ARRAYARRAY_TIME[6][8]);
    RETAINTEST_AUTO_STRUCTUREARRAYARRAY.ARRAYARRAY_STRING[6][9] := ANY_TO_STRING(RETAINTEST_AUTO_ARRAYARRAY_DINT[6][9]) + ' ' + ANY_TO_STRING(RETAINTEST_AUTO_ARRAYARRAY_TIME[6][9]);

    RETAINTEST_AUTO_STRUCTUREARRAYARRAY.ARRAYARRAY_STRING[7][0] := RETAINTEST_AUTO_STRUCTUREARRAYARRAY.ARRAYARRAY_STRING[6][0];
    RETAINTEST_AUTO_STRUCTUREARRAYARRAY.ARRAYARRAY_STRING[7][1] := RETAINTEST_AUTO_STRUCTUREARRAYARRAY.ARRAYARRAY_STRING[6][1];
    RETAINTEST_AUTO_STRUCTUREARRAYARRAY.ARRAYARRAY_STRING[7][2] := RETAINTEST_AUTO_STRUCTUREARRAYARRAY.ARRAYARRAY_STRING[6][2];
    RETAINTEST_AUTO_STRUCTUREARRAYARRAY.ARRAYARRAY_STRING[7][3] := RETAINTEST_AUTO_STRUCTUREARRAYARRAY.ARRAYARRAY_STRING[6][3];
    RETAINTEST_AUTO_STRUCTUREARRAYARRAY.ARRAYARRAY_STRING[7][4] := RETAINTEST_AUTO_STRUCTUREARRAYARRAY.ARRAYARRAY_STRING[6][4];
    RETAINTEST_AUTO_STRUCTUREARRAYARRAY.ARRAYARRAY_STRING[7][5] := RETAINTEST_AUTO_STRUCTUREARRAYARRAY.ARRAYARRAY_STRING[6][5];
    RETAINTEST_AUTO_STRUCTUREARRAYARRAY.ARRAYARRAY_STRING[7][6] := RETAINTEST_AUTO_STRUCTUREARRAYARRAY.ARRAYARRAY_STRING[6][6];
    RETAINTEST_AUTO_STRUCTUREARRAYARRAY.ARRAYARRAY_STRING[7][7] := RETAINTEST_AUTO_STRUCTUREARRAYARRAY.ARRAYARRAY_STRING[6][7];
    RETAINTEST_AUTO_STRUCTUREARRAYARRAY.ARRAYARRAY_STRING[7][8] := RETAINTEST_AUTO_STRUCTUREARRAYARRAY.ARRAYARRAY_STRING[6][8];
    RETAINTEST_AUTO_STRUCTUREARRAYARRAY.ARRAYARRAY_STRING[7][9] := RETAINTEST_AUTO_STRUCTUREARRAYARRAY.ARRAYARRAY_STRING[6][9];

    RETAINTEST_AUTO_STRUCTUREARRAYARRAY.ARRAYARRAY_TIME[0][0] := RETAINTEST_AUTO_STRUCTUREARRAYARRAY.ARRAYARRAY_TIME[0][0] + PULSE_TIME;
    RETAINTEST_AUTO_STRUCTUREARRAYARRAY.ARRAYARRAY_TIME[0][1] := RETAINTEST_AUTO_STRUCTUREARRAYARRAY.ARRAYARRAY_TIME[0][1] + PULSE_TIME;
    RETAINTEST_AUTO_STRUCTUREARRAYARRAY.ARRAYARRAY_TIME[0][2] := RETAINTEST_AUTO_STRUCTUREARRAYARRAY.ARRAYARRAY_TIME[0][2] + PULSE_TIME;
    RETAINTEST_AUTO_STRUCTUREARRAYARRAY.ARRAYARRAY_TIME[0][3] := RETAINTEST_AUTO_STRUCTUREARRAYARRAY.ARRAYARRAY_TIME[0][3] + PULSE_TIME;
    RETAINTEST_AUTO_STRUCTUREARRAYARRAY.ARRAYARRAY_TIME[0][4] := RETAINTEST_AUTO_STRUCTUREARRAYARRAY.ARRAYARRAY_TIME[0][4] + PULSE_TIME;
    RETAINTEST_AUTO_STRUCTUREARRAYARRAY.ARRAYARRAY_TIME[0][5] := RETAINTEST_AUTO_STRUCTUREARRAYARRAY.ARRAYARRAY_TIME[0][5] + PULSE_TIME;
    RETAINTEST_AUTO_STRUCTUREARRAYARRAY.ARRAYARRAY_TIME[0][6] := RETAINTEST_AUTO_STRUCTUREARRAYARRAY.ARRAYARRAY_TIME[0][6] + PULSE_TIME;
    RETAINTEST_AUTO_STRUCTUREARRAYARRAY.ARRAYARRAY_TIME[0][7] := RETAINTEST_AUTO_STRUCTUREARRAYARRAY.ARRAYARRAY_TIME[0][7] + PULSE_TIME;
    RETAINTEST_AUTO_STRUCTUREARRAYARRAY.ARRAYARRAY_TIME[0][8] := RETAINTEST_AUTO_STRUCTUREARRAYARRAY.ARRAYARRAY_TIME[0][6];
    RETAINTEST_AUTO_STRUCTUREARRAYARRAY.ARRAYARRAY_TIME[0][9] := RETAINTEST_AUTO_STRUCTUREARRAYARRAY.ARRAYARRAY_TIME[0][7];

    RETAINTEST_AUTO_STRUCTUREARRAYARRAY.ARRAYARRAY_TIME[1][0] := RETAINTEST_AUTO_STRUCTUREARRAYARRAY.ARRAYARRAY_TIME[1][0] + PULSE_TIME;
    RETAINTEST_AUTO_STRUCTUREARRAYARRAY.ARRAYARRAY_TIME[1][1] := RETAINTEST_AUTO_STRUCTUREARRAYARRAY.ARRAYARRAY_TIME[1][1] + PULSE_TIME;
    RETAINTEST_AUTO_STRUCTUREARRAYARRAY.ARRAYARRAY_TIME[1][2] := RETAINTEST_AUTO_STRUCTUREARRAYARRAY.ARRAYARRAY_TIME[1][2] + PULSE_TIME;
    RETAINTEST_AUTO_STRUCTUREARRAYARRAY.ARRAYARRAY_TIME[1][3] := RETAINTEST_AUTO_STRUCTUREARRAYARRAY.ARRAYARRAY_TIME[1][3] + PULSE_TIME;
    RETAINTEST_AUTO_STRUCTUREARRAYARRAY.ARRAYARRAY_TIME[1][4] := RETAINTEST_AUTO_STRUCTUREARRAYARRAY.ARRAYARRAY_TIME[1][4] + PULSE_TIME;
    RETAINTEST_AUTO_STRUCTUREARRAYARRAY.ARRAYARRAY_TIME[1][5] := RETAINTEST_AUTO_STRUCTUREARRAYARRAY.ARRAYARRAY_TIME[1][5] + PULSE_TIME;
    RETAINTEST_AUTO_STRUCTUREARRAYARRAY.ARRAYARRAY_TIME[1][6] := RETAINTEST_AUTO_STRUCTUREARRAYARRAY.ARRAYARRAY_TIME[1][6] + PULSE_TIME;
    RETAINTEST_AUTO_STRUCTUREARRAYARRAY.ARRAYARRAY_TIME[1][7] := RETAINTEST_AUTO_STRUCTUREARRAYARRAY.ARRAYARRAY_TIME[1][7] + PULSE_TIME;
    RETAINTEST_AUTO_STRUCTUREARRAYARRAY.ARRAYARRAY_TIME[1][8] := RETAINTEST_AUTO_STRUCTUREARRAYARRAY.ARRAYARRAY_TIME[1][6];
    RETAINTEST_AUTO_STRUCTUREARRAYARRAY.ARRAYARRAY_TIME[1][9] := RETAINTEST_AUTO_STRUCTUREARRAYARRAY.ARRAYARRAY_TIME[1][7];

    RETAINTEST_AUTO_STRUCTUREARRAYARRAY.ARRAYARRAY_TIME[2][0] := RETAINTEST_AUTO_STRUCTUREARRAYARRAY.ARRAYARRAY_TIME[2][0] + PULSE_TIME;
    RETAINTEST_AUTO_STRUCTUREARRAYARRAY.ARRAYARRAY_TIME[2][1] := RETAINTEST_AUTO_STRUCTUREARRAYARRAY.ARRAYARRAY_TIME[2][1] + PULSE_TIME;
    RETAINTEST_AUTO_STRUCTUREARRAYARRAY.ARRAYARRAY_TIME[2][2] := RETAINTEST_AUTO_STRUCTUREARRAYARRAY.ARRAYARRAY_TIME[2][2] + PULSE_TIME;
    RETAINTEST_AUTO_STRUCTUREARRAYARRAY.ARRAYARRAY_TIME[2][3] := RETAINTEST_AUTO_STRUCTUREARRAYARRAY.ARRAYARRAY_TIME[2][3] + PULSE_TIME;
    RETAINTEST_AUTO_STRUCTUREARRAYARRAY.ARRAYARRAY_TIME[2][4] := RETAINTEST_AUTO_STRUCTUREARRAYARRAY.ARRAYARRAY_TIME[2][4] + PULSE_TIME;
    RETAINTEST_AUTO_STRUCTUREARRAYARRAY.ARRAYARRAY_TIME[2][5] := RETAINTEST_AUTO_STRUCTUREARRAYARRAY.ARRAYARRAY_TIME[2][5] + PULSE_TIME;
    RETAINTEST_AUTO_STRUCTUREARRAYARRAY.ARRAYARRAY_TIME[2][6] := RETAINTEST_AUTO_STRUCTUREARRAYARRAY.ARRAYARRAY_TIME[2][6] + PULSE_TIME;
    RETAINTEST_AUTO_STRUCTUREARRAYARRAY.ARRAYARRAY_TIME[2][7] := RETAINTEST_AUTO_STRUCTUREARRAYARRAY.ARRAYARRAY_TIME[2][7] + PULSE_TIME;
    RETAINTEST_AUTO_STRUCTUREARRAYARRAY.ARRAYARRAY_TIME[2][8] := RETAINTEST_AUTO_STRUCTUREARRAYARRAY.ARRAYARRAY_TIME[2][8] + PULSE_TIME;
    RETAINTEST_AUTO_STRUCTUREARRAYARRAY.ARRAYARRAY_TIME[2][9] := RETAINTEST_AUTO_STRUCTUREARRAYARRAY.ARRAYARRAY_TIME[2][9] + PULSE_TIME;

    RETAINTEST_AUTO_STRUCTUREARRAYARRAY.ARRAYARRAY_TIME[3][0] := RETAINTEST_AUTO_STRUCTUREARRAYARRAY.ARRAYARRAY_TIME[3][0] + PULSE_TIME;
    RETAINTEST_AUTO_STRUCTUREARRAYARRAY.ARRAYARRAY_TIME[3][1] := RETAINTEST_AUTO_STRUCTUREARRAYARRAY.ARRAYARRAY_TIME[3][1] + PULSE_TIME;
    RETAINTEST_AUTO_STRUCTUREARRAYARRAY.ARRAYARRAY_TIME[3][2] := RETAINTEST_AUTO_STRUCTUREARRAYARRAY.ARRAYARRAY_TIME[3][2] + PULSE_TIME;
    RETAINTEST_AUTO_STRUCTUREARRAYARRAY.ARRAYARRAY_TIME[3][3] := RETAINTEST_AUTO_STRUCTUREARRAYARRAY.ARRAYARRAY_TIME[3][3] + PULSE_TIME;
    RETAINTEST_AUTO_STRUCTUREARRAYARRAY.ARRAYARRAY_TIME[3][4] := RETAINTEST_AUTO_STRUCTUREARRAYARRAY.ARRAYARRAY_TIME[3][4] + PULSE_TIME;
    RETAINTEST_AUTO_STRUCTUREARRAYARRAY.ARRAYARRAY_TIME[3][5] := RETAINTEST_AUTO_STRUCTUREARRAYARRAY.ARRAYARRAY_TIME[3][5] + PULSE_TIME;
    RETAINTEST_AUTO_STRUCTUREARRAYARRAY.ARRAYARRAY_TIME[3][6] := RETAINTEST_AUTO_STRUCTUREARRAYARRAY.ARRAYARRAY_TIME[3][6] + PULSE_TIME;
    RETAINTEST_AUTO_STRUCTUREARRAYARRAY.ARRAYARRAY_TIME[3][7] := RETAINTEST_AUTO_STRUCTUREARRAYARRAY.ARRAYARRAY_TIME[3][7] + PULSE_TIME;
    RETAINTEST_AUTO_STRUCTUREARRAYARRAY.ARRAYARRAY_TIME[3][8] := RETAINTEST_AUTO_STRUCTUREARRAYARRAY.ARRAYARRAY_TIME[3][8] + PULSE_TIME;
    RETAINTEST_AUTO_STRUCTUREARRAYARRAY.ARRAYARRAY_TIME[3][9] := RETAINTEST_AUTO_STRUCTUREARRAYARRAY.ARRAYARRAY_TIME[3][9] + PULSE_TIME;

    RETAINTEST_AUTO_STRUCTUREARRAYARRAY.ARRAYARRAY_TIME[4][0] := RETAINTEST_AUTO_STRUCTUREARRAYARRAY.ARRAYARRAY_TIME[4][0] + PULSE_TIME;
    RETAINTEST_AUTO_STRUCTUREARRAYARRAY.ARRAYARRAY_TIME[4][1] := RETAINTEST_AUTO_STRUCTUREARRAYARRAY.ARRAYARRAY_TIME[4][1] + PULSE_TIME;
    RETAINTEST_AUTO_STRUCTUREARRAYARRAY.ARRAYARRAY_TIME[4][2] := RETAINTEST_AUTO_STRUCTUREARRAYARRAY.ARRAYARRAY_TIME[4][2] + PULSE_TIME;
    RETAINTEST_AUTO_STRUCTUREARRAYARRAY.ARRAYARRAY_TIME[4][3] := RETAINTEST_AUTO_STRUCTUREARRAYARRAY.ARRAYARRAY_TIME[4][3] + PULSE_TIME;
    RETAINTEST_AUTO_STRUCTUREARRAYARRAY.ARRAYARRAY_TIME[4][4] := RETAINTEST_AUTO_STRUCTUREARRAYARRAY.ARRAYARRAY_TIME[4][4] + PULSE_TIME;
    RETAINTEST_AUTO_STRUCTUREARRAYARRAY.ARRAYARRAY_TIME[4][5] := RETAINTEST_AUTO_STRUCTUREARRAYARRAY.ARRAYARRAY_TIME[4][5] + PULSE_TIME;
    RETAINTEST_AUTO_STRUCTUREARRAYARRAY.ARRAYARRAY_TIME[4][6] := RETAINTEST_AUTO_STRUCTUREARRAYARRAY.ARRAYARRAY_TIME[4][6] + PULSE_TIME;
    RETAINTEST_AUTO_STRUCTUREARRAYARRAY.ARRAYARRAY_TIME[4][7] := RETAINTEST_AUTO_STRUCTUREARRAYARRAY.ARRAYARRAY_TIME[4][7] + PULSE_TIME;
    RETAINTEST_AUTO_STRUCTUREARRAYARRAY.ARRAYARRAY_TIME[4][8] := RETAINTEST_AUTO_STRUCTUREARRAYARRAY.ARRAYARRAY_TIME[4][8] + PULSE_TIME;
    RETAINTEST_AUTO_STRUCTUREARRAYARRAY.ARRAYARRAY_TIME[4][9] := RETAINTEST_AUTO_STRUCTUREARRAYARRAY.ARRAYARRAY_TIME[4][9] + PULSE_TIME;

    RETAINTEST_AUTO_STRUCTUREARRAYARRAY.ARRAYARRAY_TIME[5][0] := RETAINTEST_AUTO_STRUCTUREARRAYARRAY.ARRAYARRAY_TIME[5][0] + PULSE_TIME;
    RETAINTEST_AUTO_STRUCTUREARRAYARRAY.ARRAYARRAY_TIME[5][1] := RETAINTEST_AUTO_STRUCTUREARRAYARRAY.ARRAYARRAY_TIME[5][1] + PULSE_TIME;
    RETAINTEST_AUTO_STRUCTUREARRAYARRAY.ARRAYARRAY_TIME[5][2] := RETAINTEST_AUTO_STRUCTUREARRAYARRAY.ARRAYARRAY_TIME[5][2] + PULSE_TIME;
    RETAINTEST_AUTO_STRUCTUREARRAYARRAY.ARRAYARRAY_TIME[5][3] := RETAINTEST_AUTO_STRUCTUREARRAYARRAY.ARRAYARRAY_TIME[5][3] + PULSE_TIME;
    RETAINTEST_AUTO_STRUCTUREARRAYARRAY.ARRAYARRAY_TIME[5][4] := RETAINTEST_AUTO_STRUCTUREARRAYARRAY.ARRAYARRAY_TIME[5][4] + PULSE_TIME;
    RETAINTEST_AUTO_STRUCTUREARRAYARRAY.ARRAYARRAY_TIME[5][5] := RETAINTEST_AUTO_STRUCTUREARRAYARRAY.ARRAYARRAY_TIME[5][5] + PULSE_TIME;
    RETAINTEST_AUTO_STRUCTUREARRAYARRAY.ARRAYARRAY_TIME[5][6] := RETAINTEST_AUTO_STRUCTUREARRAYARRAY.ARRAYARRAY_TIME[5][6] + PULSE_TIME;
    RETAINTEST_AUTO_STRUCTUREARRAYARRAY.ARRAYARRAY_TIME[5][7] := RETAINTEST_AUTO_STRUCTUREARRAYARRAY.ARRAYARRAY_TIME[5][7] + PULSE_TIME;
    RETAINTEST_AUTO_STRUCTUREARRAYARRAY.ARRAYARRAY_TIME[5][8] := RETAINTEST_AUTO_STRUCTUREARRAYARRAY.ARRAYARRAY_TIME[5][8] + PULSE_TIME;
    RETAINTEST_AUTO_STRUCTUREARRAYARRAY.ARRAYARRAY_TIME[5][9] := RETAINTEST_AUTO_STRUCTUREARRAYARRAY.ARRAYARRAY_TIME[5][9] + PULSE_TIME;

    RETAINTEST_AUTO_STRUCTUREARRAYARRAY.ARRAYARRAY_TIME[6][0] := RETAINTEST_AUTO_STRUCTUREARRAYARRAY.ARRAYARRAY_TIME[6][0] + PULSE_TIME;
    RETAINTEST_AUTO_STRUCTUREARRAYARRAY.ARRAYARRAY_TIME[6][1] := RETAINTEST_AUTO_STRUCTUREARRAYARRAY.ARRAYARRAY_TIME[6][1] + PULSE_TIME;
    RETAINTEST_AUTO_STRUCTUREARRAYARRAY.ARRAYARRAY_TIME[6][2] := RETAINTEST_AUTO_STRUCTUREARRAYARRAY.ARRAYARRAY_TIME[6][2] + PULSE_TIME;
    RETAINTEST_AUTO_STRUCTUREARRAYARRAY.ARRAYARRAY_TIME[6][3] := RETAINTEST_AUTO_STRUCTUREARRAYARRAY.ARRAYARRAY_TIME[6][3] + PULSE_TIME;
    RETAINTEST_AUTO_STRUCTUREARRAYARRAY.ARRAYARRAY_TIME[6][4] := RETAINTEST_AUTO_STRUCTUREARRAYARRAY.ARRAYARRAY_TIME[6][4] + PULSE_TIME;
    RETAINTEST_AUTO_STRUCTUREARRAYARRAY.ARRAYARRAY_TIME[6][5] := RETAINTEST_AUTO_STRUCTUREARRAYARRAY.ARRAYARRAY_TIME[6][5] + PULSE_TIME;
    RETAINTEST_AUTO_STRUCTUREARRAYARRAY.ARRAYARRAY_TIME[6][6] := RETAINTEST_AUTO_STRUCTUREARRAYARRAY.ARRAYARRAY_TIME[6][6] + PULSE_TIME;
    RETAINTEST_AUTO_STRUCTUREARRAYARRAY.ARRAYARRAY_TIME[6][7] := RETAINTEST_AUTO_STRUCTUREARRAYARRAY.ARRAYARRAY_TIME[6][7] + PULSE_TIME;
    RETAINTEST_AUTO_STRUCTUREARRAYARRAY.ARRAYARRAY_TIME[6][8] := RETAINTEST_AUTO_STRUCTUREARRAYARRAY.ARRAYARRAY_TIME[6][8] + PULSE_TIME;
    RETAINTEST_AUTO_STRUCTUREARRAYARRAY.ARRAYARRAY_TIME[6][9] := RETAINTEST_AUTO_STRUCTUREARRAYARRAY.ARRAYARRAY_TIME[6][9] + PULSE_TIME;

    RETAINTEST_AUTO_STRUCTUREARRAYARRAY.ARRAYARRAY_TIME[7][0] := RETAINTEST_AUTO_STRUCTUREARRAYARRAY.ARRAYARRAY_TIME[6][0];
    RETAINTEST_AUTO_STRUCTUREARRAYARRAY.ARRAYARRAY_TIME[7][1] := RETAINTEST_AUTO_STRUCTUREARRAYARRAY.ARRAYARRAY_TIME[6][1];
    RETAINTEST_AUTO_STRUCTUREARRAYARRAY.ARRAYARRAY_TIME[7][2] := RETAINTEST_AUTO_STRUCTUREARRAYARRAY.ARRAYARRAY_TIME[6][2];
    RETAINTEST_AUTO_STRUCTUREARRAYARRAY.ARRAYARRAY_TIME[7][3] := RETAINTEST_AUTO_STRUCTUREARRAYARRAY.ARRAYARRAY_TIME[6][3];
    RETAINTEST_AUTO_STRUCTUREARRAYARRAY.ARRAYARRAY_TIME[7][4] := RETAINTEST_AUTO_STRUCTUREARRAYARRAY.ARRAYARRAY_TIME[6][4];
    RETAINTEST_AUTO_STRUCTUREARRAYARRAY.ARRAYARRAY_TIME[7][5] := RETAINTEST_AUTO_STRUCTUREARRAYARRAY.ARRAYARRAY_TIME[6][5];
    RETAINTEST_AUTO_STRUCTUREARRAYARRAY.ARRAYARRAY_TIME[7][6] := RETAINTEST_AUTO_STRUCTUREARRAYARRAY.ARRAYARRAY_TIME[6][6];
    RETAINTEST_AUTO_STRUCTUREARRAYARRAY.ARRAYARRAY_TIME[7][7] := RETAINTEST_AUTO_STRUCTUREARRAYARRAY.ARRAYARRAY_TIME[6][7];
    RETAINTEST_AUTO_STRUCTUREARRAYARRAY.ARRAYARRAY_TIME[7][8] := RETAINTEST_AUTO_STRUCTUREARRAYARRAY.ARRAYARRAY_TIME[6][8];
    RETAINTEST_AUTO_STRUCTUREARRAYARRAY.ARRAYARRAY_TIME[7][9] := RETAINTEST_AUTO_STRUCTUREARRAYARRAY.ARRAYARRAY_TIME[6][9];

    RETAINTEST_AUTO_STRUCTUREARRAYARRAY.ARRAYARRAY_UDINT[0][0] := RETAINTEST_AUTO_STRUCTUREARRAYARRAY.ARRAYARRAY_UDINT[0][0] + 1;
    RETAINTEST_AUTO_STRUCTUREARRAYARRAY.ARRAYARRAY_UDINT[0][1] := RETAINTEST_AUTO_STRUCTUREARRAYARRAY.ARRAYARRAY_UDINT[0][1] + 1;
    RETAINTEST_AUTO_STRUCTUREARRAYARRAY.ARRAYARRAY_UDINT[0][2] := RETAINTEST_AUTO_STRUCTUREARRAYARRAY.ARRAYARRAY_UDINT[0][2] + 1;
    RETAINTEST_AUTO_STRUCTUREARRAYARRAY.ARRAYARRAY_UDINT[0][3] := RETAINTEST_AUTO_STRUCTUREARRAYARRAY.ARRAYARRAY_UDINT[0][3] + 1;
    RETAINTEST_AUTO_STRUCTUREARRAYARRAY.ARRAYARRAY_UDINT[0][4] := RETAINTEST_AUTO_STRUCTUREARRAYARRAY.ARRAYARRAY_UDINT[0][4] + 1;
    RETAINTEST_AUTO_STRUCTUREARRAYARRAY.ARRAYARRAY_UDINT[0][5] := RETAINTEST_AUTO_STRUCTUREARRAYARRAY.ARRAYARRAY_UDINT[0][5] + 1;
    RETAINTEST_AUTO_STRUCTUREARRAYARRAY.ARRAYARRAY_UDINT[0][6] := RETAINTEST_AUTO_STRUCTUREARRAYARRAY.ARRAYARRAY_UDINT[0][6] + 1;
    RETAINTEST_AUTO_STRUCTUREARRAYARRAY.ARRAYARRAY_UDINT[0][7] := RETAINTEST_AUTO_STRUCTUREARRAYARRAY.ARRAYARRAY_UDINT[0][7] + 1;
    RETAINTEST_AUTO_STRUCTUREARRAYARRAY.ARRAYARRAY_UDINT[0][8] := RETAINTEST_AUTO_STRUCTUREARRAYARRAY.ARRAYARRAY_UDINT[0][6];
    RETAINTEST_AUTO_STRUCTUREARRAYARRAY.ARRAYARRAY_UDINT[0][9] := RETAINTEST_AUTO_STRUCTUREARRAYARRAY.ARRAYARRAY_UDINT[0][7];

    RETAINTEST_AUTO_STRUCTUREARRAYARRAY.ARRAYARRAY_UDINT[1][0] := RETAINTEST_AUTO_STRUCTUREARRAYARRAY.ARRAYARRAY_UDINT[1][0] + 1;
    RETAINTEST_AUTO_STRUCTUREARRAYARRAY.ARRAYARRAY_UDINT[1][1] := RETAINTEST_AUTO_STRUCTUREARRAYARRAY.ARRAYARRAY_UDINT[1][1] + 1;
    RETAINTEST_AUTO_STRUCTUREARRAYARRAY.ARRAYARRAY_UDINT[1][2] := RETAINTEST_AUTO_STRUCTUREARRAYARRAY.ARRAYARRAY_UDINT[1][2] + 1;
    RETAINTEST_AUTO_STRUCTUREARRAYARRAY.ARRAYARRAY_UDINT[1][3] := RETAINTEST_AUTO_STRUCTUREARRAYARRAY.ARRAYARRAY_UDINT[1][3] + 1;
    RETAINTEST_AUTO_STRUCTUREARRAYARRAY.ARRAYARRAY_UDINT[1][4] := RETAINTEST_AUTO_STRUCTUREARRAYARRAY.ARRAYARRAY_UDINT[1][4] + 1;
    RETAINTEST_AUTO_STRUCTUREARRAYARRAY.ARRAYARRAY_UDINT[1][5] := RETAINTEST_AUTO_STRUCTUREARRAYARRAY.ARRAYARRAY_UDINT[1][5] + 1;
    RETAINTEST_AUTO_STRUCTUREARRAYARRAY.ARRAYARRAY_UDINT[1][6] := RETAINTEST_AUTO_STRUCTUREARRAYARRAY.ARRAYARRAY_UDINT[1][6] + 1;
    RETAINTEST_AUTO_STRUCTUREARRAYARRAY.ARRAYARRAY_UDINT[1][7] := RETAINTEST_AUTO_STRUCTUREARRAYARRAY.ARRAYARRAY_UDINT[1][7] + 1;
    RETAINTEST_AUTO_STRUCTUREARRAYARRAY.ARRAYARRAY_UDINT[1][8] := RETAINTEST_AUTO_STRUCTUREARRAYARRAY.ARRAYARRAY_UDINT[1][6];
    RETAINTEST_AUTO_STRUCTUREARRAYARRAY.ARRAYARRAY_UDINT[1][9] := RETAINTEST_AUTO_STRUCTUREARRAYARRAY.ARRAYARRAY_UDINT[1][7];

    RETAINTEST_AUTO_STRUCTUREARRAYARRAY.ARRAYARRAY_UDINT[2][0] := RETAINTEST_AUTO_STRUCTUREARRAYARRAY.ARRAYARRAY_UDINT[2][0] + 1;
    RETAINTEST_AUTO_STRUCTUREARRAYARRAY.ARRAYARRAY_UDINT[2][1] := RETAINTEST_AUTO_STRUCTUREARRAYARRAY.ARRAYARRAY_UDINT[2][1] + 1;
    RETAINTEST_AUTO_STRUCTUREARRAYARRAY.ARRAYARRAY_UDINT[2][2] := RETAINTEST_AUTO_STRUCTUREARRAYARRAY.ARRAYARRAY_UDINT[2][2] + 1;
    RETAINTEST_AUTO_STRUCTUREARRAYARRAY.ARRAYARRAY_UDINT[2][3] := RETAINTEST_AUTO_STRUCTUREARRAYARRAY.ARRAYARRAY_UDINT[2][3] + 1;
    RETAINTEST_AUTO_STRUCTUREARRAYARRAY.ARRAYARRAY_UDINT[2][4] := RETAINTEST_AUTO_STRUCTUREARRAYARRAY.ARRAYARRAY_UDINT[2][4] + 1;
    RETAINTEST_AUTO_STRUCTUREARRAYARRAY.ARRAYARRAY_UDINT[2][5] := RETAINTEST_AUTO_STRUCTUREARRAYARRAY.ARRAYARRAY_UDINT[2][5] + 1;
    RETAINTEST_AUTO_STRUCTUREARRAYARRAY.ARRAYARRAY_UDINT[2][6] := RETAINTEST_AUTO_STRUCTUREARRAYARRAY.ARRAYARRAY_UDINT[2][6] + 1;
    RETAINTEST_AUTO_STRUCTUREARRAYARRAY.ARRAYARRAY_UDINT[2][7] := RETAINTEST_AUTO_STRUCTUREARRAYARRAY.ARRAYARRAY_UDINT[2][7] + 1;
    RETAINTEST_AUTO_STRUCTUREARRAYARRAY.ARRAYARRAY_UDINT[2][8] := RETAINTEST_AUTO_STRUCTUREARRAYARRAY.ARRAYARRAY_UDINT[2][8] + 1;
    RETAINTEST_AUTO_STRUCTUREARRAYARRAY.ARRAYARRAY_UDINT[2][9] := RETAINTEST_AUTO_STRUCTUREARRAYARRAY.ARRAYARRAY_UDINT[2][9] + 1;

    RETAINTEST_AUTO_STRUCTUREARRAYARRAY.ARRAYARRAY_UDINT[3][0] := RETAINTEST_AUTO_STRUCTUREARRAYARRAY.ARRAYARRAY_UDINT[3][0] + 1;
    RETAINTEST_AUTO_STRUCTUREARRAYARRAY.ARRAYARRAY_UDINT[3][1] := RETAINTEST_AUTO_STRUCTUREARRAYARRAY.ARRAYARRAY_UDINT[3][1] + 1;
    RETAINTEST_AUTO_STRUCTUREARRAYARRAY.ARRAYARRAY_UDINT[3][2] := RETAINTEST_AUTO_STRUCTUREARRAYARRAY.ARRAYARRAY_UDINT[3][2] + 1;
    RETAINTEST_AUTO_STRUCTUREARRAYARRAY.ARRAYARRAY_UDINT[3][3] := RETAINTEST_AUTO_STRUCTUREARRAYARRAY.ARRAYARRAY_UDINT[3][3] + 1;
    RETAINTEST_AUTO_STRUCTUREARRAYARRAY.ARRAYARRAY_UDINT[3][4] := RETAINTEST_AUTO_STRUCTUREARRAYARRAY.ARRAYARRAY_UDINT[3][4] + 1;
    RETAINTEST_AUTO_STRUCTUREARRAYARRAY.ARRAYARRAY_UDINT[3][5] := RETAINTEST_AUTO_STRUCTUREARRAYARRAY.ARRAYARRAY_UDINT[3][5] + 1;
    RETAINTEST_AUTO_STRUCTUREARRAYARRAY.ARRAYARRAY_UDINT[3][6] := RETAINTEST_AUTO_STRUCTUREARRAYARRAY.ARRAYARRAY_UDINT[3][6] + 1;
    RETAINTEST_AUTO_STRUCTUREARRAYARRAY.ARRAYARRAY_UDINT[3][7] := RETAINTEST_AUTO_STRUCTUREARRAYARRAY.ARRAYARRAY_UDINT[3][7] + 1;
    RETAINTEST_AUTO_STRUCTUREARRAYARRAY.ARRAYARRAY_UDINT[3][8] := RETAINTEST_AUTO_STRUCTUREARRAYARRAY.ARRAYARRAY_UDINT[3][8] + 1;
    RETAINTEST_AUTO_STRUCTUREARRAYARRAY.ARRAYARRAY_UDINT[3][9] := RETAINTEST_AUTO_STRUCTUREARRAYARRAY.ARRAYARRAY_UDINT[3][9] + 1;

    RETAINTEST_AUTO_STRUCTUREARRAYARRAY.ARRAYARRAY_UDINT[4][0] := RETAINTEST_AUTO_STRUCTUREARRAYARRAY.ARRAYARRAY_UDINT[4][0] + 1;
    RETAINTEST_AUTO_STRUCTUREARRAYARRAY.ARRAYARRAY_UDINT[4][1] := RETAINTEST_AUTO_STRUCTUREARRAYARRAY.ARRAYARRAY_UDINT[4][1] + 1;
    RETAINTEST_AUTO_STRUCTUREARRAYARRAY.ARRAYARRAY_UDINT[4][2] := RETAINTEST_AUTO_STRUCTUREARRAYARRAY.ARRAYARRAY_UDINT[4][2] + 1;
    RETAINTEST_AUTO_STRUCTUREARRAYARRAY.ARRAYARRAY_UDINT[4][3] := RETAINTEST_AUTO_STRUCTUREARRAYARRAY.ARRAYARRAY_UDINT[4][3] + 1;
    RETAINTEST_AUTO_STRUCTUREARRAYARRAY.ARRAYARRAY_UDINT[4][4] := RETAINTEST_AUTO_STRUCTUREARRAYARRAY.ARRAYARRAY_UDINT[4][4] + 1;
    RETAINTEST_AUTO_STRUCTUREARRAYARRAY.ARRAYARRAY_UDINT[4][5] := RETAINTEST_AUTO_STRUCTUREARRAYARRAY.ARRAYARRAY_UDINT[4][5] + 1;
    RETAINTEST_AUTO_STRUCTUREARRAYARRAY.ARRAYARRAY_UDINT[4][6] := RETAINTEST_AUTO_STRUCTUREARRAYARRAY.ARRAYARRAY_UDINT[4][6] + 1;
    RETAINTEST_AUTO_STRUCTUREARRAYARRAY.ARRAYARRAY_UDINT[4][7] := RETAINTEST_AUTO_STRUCTUREARRAYARRAY.ARRAYARRAY_UDINT[4][7] + 1;
    RETAINTEST_AUTO_STRUCTUREARRAYARRAY.ARRAYARRAY_UDINT[4][8] := RETAINTEST_AUTO_STRUCTUREARRAYARRAY.ARRAYARRAY_UDINT[4][8] + 1;
    RETAINTEST_AUTO_STRUCTUREARRAYARRAY.ARRAYARRAY_UDINT[4][9] := RETAINTEST_AUTO_STRUCTUREARRAYARRAY.ARRAYARRAY_UDINT[4][9] + 1;

    RETAINTEST_AUTO_STRUCTUREARRAYARRAY.ARRAYARRAY_UDINT[5][0] := RETAINTEST_AUTO_STRUCTUREARRAYARRAY.ARRAYARRAY_UDINT[5][0] + 1;
    RETAINTEST_AUTO_STRUCTUREARRAYARRAY.ARRAYARRAY_UDINT[5][1] := RETAINTEST_AUTO_STRUCTUREARRAYARRAY.ARRAYARRAY_UDINT[5][1] + 1;
    RETAINTEST_AUTO_STRUCTUREARRAYARRAY.ARRAYARRAY_UDINT[5][2] := RETAINTEST_AUTO_STRUCTUREARRAYARRAY.ARRAYARRAY_UDINT[5][2] + 1;
    RETAINTEST_AUTO_STRUCTUREARRAYARRAY.ARRAYARRAY_UDINT[5][3] := RETAINTEST_AUTO_STRUCTUREARRAYARRAY.ARRAYARRAY_UDINT[5][3] + 1;
    RETAINTEST_AUTO_STRUCTUREARRAYARRAY.ARRAYARRAY_UDINT[5][4] := RETAINTEST_AUTO_STRUCTUREARRAYARRAY.ARRAYARRAY_UDINT[5][4] + 1;
    RETAINTEST_AUTO_STRUCTUREARRAYARRAY.ARRAYARRAY_UDINT[5][5] := RETAINTEST_AUTO_STRUCTUREARRAYARRAY.ARRAYARRAY_UDINT[5][5] + 1;
    RETAINTEST_AUTO_STRUCTUREARRAYARRAY.ARRAYARRAY_UDINT[5][6] := RETAINTEST_AUTO_STRUCTUREARRAYARRAY.ARRAYARRAY_UDINT[5][6] + 1;
    RETAINTEST_AUTO_STRUCTUREARRAYARRAY.ARRAYARRAY_UDINT[5][7] := RETAINTEST_AUTO_STRUCTUREARRAYARRAY.ARRAYARRAY_UDINT[5][7] + 1;
    RETAINTEST_AUTO_STRUCTUREARRAYARRAY.ARRAYARRAY_UDINT[5][8] := RETAINTEST_AUTO_STRUCTUREARRAYARRAY.ARRAYARRAY_UDINT[5][8] + 1;
    RETAINTEST_AUTO_STRUCTUREARRAYARRAY.ARRAYARRAY_UDINT[5][9] := RETAINTEST_AUTO_STRUCTUREARRAYARRAY.ARRAYARRAY_UDINT[5][9] + 1;

    RETAINTEST_AUTO_STRUCTUREARRAYARRAY.ARRAYARRAY_UDINT[6][0] := RETAINTEST_AUTO_STRUCTUREARRAYARRAY.ARRAYARRAY_UDINT[6][0] + 1;
    RETAINTEST_AUTO_STRUCTUREARRAYARRAY.ARRAYARRAY_UDINT[6][1] := RETAINTEST_AUTO_STRUCTUREARRAYARRAY.ARRAYARRAY_UDINT[6][1] + 1;
    RETAINTEST_AUTO_STRUCTUREARRAYARRAY.ARRAYARRAY_UDINT[6][2] := RETAINTEST_AUTO_STRUCTUREARRAYARRAY.ARRAYARRAY_UDINT[6][2] + 1;
    RETAINTEST_AUTO_STRUCTUREARRAYARRAY.ARRAYARRAY_UDINT[6][3] := RETAINTEST_AUTO_STRUCTUREARRAYARRAY.ARRAYARRAY_UDINT[6][3] + 1;
    RETAINTEST_AUTO_STRUCTUREARRAYARRAY.ARRAYARRAY_UDINT[6][4] := RETAINTEST_AUTO_STRUCTUREARRAYARRAY.ARRAYARRAY_UDINT[6][4] + 1;
    RETAINTEST_AUTO_STRUCTUREARRAYARRAY.ARRAYARRAY_UDINT[6][5] := RETAINTEST_AUTO_STRUCTUREARRAYARRAY.ARRAYARRAY_UDINT[6][5] + 1;
    RETAINTEST_AUTO_STRUCTUREARRAYARRAY.ARRAYARRAY_UDINT[6][6] := RETAINTEST_AUTO_STRUCTUREARRAYARRAY.ARRAYARRAY_UDINT[6][6] + 1;
    RETAINTEST_AUTO_STRUCTUREARRAYARRAY.ARRAYARRAY_UDINT[6][7] := RETAINTEST_AUTO_STRUCTUREARRAYARRAY.ARRAYARRAY_UDINT[6][7] + 1;
    RETAINTEST_AUTO_STRUCTUREARRAYARRAY.ARRAYARRAY_UDINT[6][8] := RETAINTEST_AUTO_STRUCTUREARRAYARRAY.ARRAYARRAY_UDINT[6][8] + 1;
    RETAINTEST_AUTO_STRUCTUREARRAYARRAY.ARRAYARRAY_UDINT[6][9] := RETAINTEST_AUTO_STRUCTUREARRAYARRAY.ARRAYARRAY_UDINT[6][9] + 1;

    RETAINTEST_AUTO_STRUCTUREARRAYARRAY.ARRAYARRAY_UDINT[7][0] := RETAINTEST_AUTO_STRUCTUREARRAYARRAY.ARRAYARRAY_UDINT[6][0];
    RETAINTEST_AUTO_STRUCTUREARRAYARRAY.ARRAYARRAY_UDINT[7][1] := RETAINTEST_AUTO_STRUCTUREARRAYARRAY.ARRAYARRAY_UDINT[6][1];
    RETAINTEST_AUTO_STRUCTUREARRAYARRAY.ARRAYARRAY_UDINT[7][2] := RETAINTEST_AUTO_STRUCTUREARRAYARRAY.ARRAYARRAY_UDINT[6][2];
    RETAINTEST_AUTO_STRUCTUREARRAYARRAY.ARRAYARRAY_UDINT[7][3] := RETAINTEST_AUTO_STRUCTUREARRAYARRAY.ARRAYARRAY_UDINT[6][3];
    RETAINTEST_AUTO_STRUCTUREARRAYARRAY.ARRAYARRAY_UDINT[7][4] := RETAINTEST_AUTO_STRUCTUREARRAYARRAY.ARRAYARRAY_UDINT[6][4];
    RETAINTEST_AUTO_STRUCTUREARRAYARRAY.ARRAYARRAY_UDINT[7][5] := RETAINTEST_AUTO_STRUCTUREARRAYARRAY.ARRAYARRAY_UDINT[6][5];
    RETAINTEST_AUTO_STRUCTUREARRAYARRAY.ARRAYARRAY_UDINT[7][6] := RETAINTEST_AUTO_STRUCTUREARRAYARRAY.ARRAYARRAY_UDINT[6][6];
    RETAINTEST_AUTO_STRUCTUREARRAYARRAY.ARRAYARRAY_UDINT[7][7] := RETAINTEST_AUTO_STRUCTUREARRAYARRAY.ARRAYARRAY_UDINT[6][7];
    RETAINTEST_AUTO_STRUCTUREARRAYARRAY.ARRAYARRAY_UDINT[7][8] := RETAINTEST_AUTO_STRUCTUREARRAYARRAY.ARRAYARRAY_UDINT[6][8];
    RETAINTEST_AUTO_STRUCTUREARRAYARRAY.ARRAYARRAY_UDINT[7][9] := RETAINTEST_AUTO_STRUCTUREARRAYARRAY.ARRAYARRAY_UDINT[6][9];

    RETAINTEST_AUTO_STRUCTUREARRAYARRAY.ARRAYARRAY_UINT[0][0] := RETAINTEST_AUTO_STRUCTUREARRAYARRAY.ARRAYARRAY_UINT[0][0] + 1;
    RETAINTEST_AUTO_STRUCTUREARRAYARRAY.ARRAYARRAY_UINT[0][1] := RETAINTEST_AUTO_STRUCTUREARRAYARRAY.ARRAYARRAY_UINT[0][1] + 1;
    RETAINTEST_AUTO_STRUCTUREARRAYARRAY.ARRAYARRAY_UINT[0][2] := RETAINTEST_AUTO_STRUCTUREARRAYARRAY.ARRAYARRAY_UINT[0][2] + 1;
    RETAINTEST_AUTO_STRUCTUREARRAYARRAY.ARRAYARRAY_UINT[0][3] := RETAINTEST_AUTO_STRUCTUREARRAYARRAY.ARRAYARRAY_UINT[0][3] + 1;
    RETAINTEST_AUTO_STRUCTUREARRAYARRAY.ARRAYARRAY_UINT[0][4] := RETAINTEST_AUTO_STRUCTUREARRAYARRAY.ARRAYARRAY_UINT[0][4] + 1;
    RETAINTEST_AUTO_STRUCTUREARRAYARRAY.ARRAYARRAY_UINT[0][5] := RETAINTEST_AUTO_STRUCTUREARRAYARRAY.ARRAYARRAY_UINT[0][5] + 1;
    RETAINTEST_AUTO_STRUCTUREARRAYARRAY.ARRAYARRAY_UINT[0][6] := RETAINTEST_AUTO_STRUCTUREARRAYARRAY.ARRAYARRAY_UINT[0][6] + 1;
    RETAINTEST_AUTO_STRUCTUREARRAYARRAY.ARRAYARRAY_UINT[0][7] := RETAINTEST_AUTO_STRUCTUREARRAYARRAY.ARRAYARRAY_UINT[0][7] + 1;
    RETAINTEST_AUTO_STRUCTUREARRAYARRAY.ARRAYARRAY_UINT[0][8] := RETAINTEST_AUTO_STRUCTUREARRAYARRAY.ARRAYARRAY_UINT[0][6];
    RETAINTEST_AUTO_STRUCTUREARRAYARRAY.ARRAYARRAY_UINT[0][9] := RETAINTEST_AUTO_STRUCTUREARRAYARRAY.ARRAYARRAY_UINT[0][7];

    RETAINTEST_AUTO_STRUCTUREARRAYARRAY.ARRAYARRAY_UINT[1][0] := RETAINTEST_AUTO_STRUCTUREARRAYARRAY.ARRAYARRAY_UINT[1][0] + 1;
    RETAINTEST_AUTO_STRUCTUREARRAYARRAY.ARRAYARRAY_UINT[1][1] := RETAINTEST_AUTO_STRUCTUREARRAYARRAY.ARRAYARRAY_UINT[1][1] + 1;
    RETAINTEST_AUTO_STRUCTUREARRAYARRAY.ARRAYARRAY_UINT[1][2] := RETAINTEST_AUTO_STRUCTUREARRAYARRAY.ARRAYARRAY_UINT[1][2] + 1;
    RETAINTEST_AUTO_STRUCTUREARRAYARRAY.ARRAYARRAY_UINT[1][3] := RETAINTEST_AUTO_STRUCTUREARRAYARRAY.ARRAYARRAY_UINT[1][3] + 1;
    RETAINTEST_AUTO_STRUCTUREARRAYARRAY.ARRAYARRAY_UINT[1][4] := RETAINTEST_AUTO_STRUCTUREARRAYARRAY.ARRAYARRAY_UINT[1][4] + 1;
    RETAINTEST_AUTO_STRUCTUREARRAYARRAY.ARRAYARRAY_UINT[1][5] := RETAINTEST_AUTO_STRUCTUREARRAYARRAY.ARRAYARRAY_UINT[1][5] + 1;
    RETAINTEST_AUTO_STRUCTUREARRAYARRAY.ARRAYARRAY_UINT[1][6] := RETAINTEST_AUTO_STRUCTUREARRAYARRAY.ARRAYARRAY_UINT[1][6] + 1;
    RETAINTEST_AUTO_STRUCTUREARRAYARRAY.ARRAYARRAY_UINT[1][7] := RETAINTEST_AUTO_STRUCTUREARRAYARRAY.ARRAYARRAY_UINT[1][7] + 1;
    RETAINTEST_AUTO_STRUCTUREARRAYARRAY.ARRAYARRAY_UINT[1][8] := RETAINTEST_AUTO_STRUCTUREARRAYARRAY.ARRAYARRAY_UINT[1][6];
    RETAINTEST_AUTO_STRUCTUREARRAYARRAY.ARRAYARRAY_UINT[1][9] := RETAINTEST_AUTO_STRUCTUREARRAYARRAY.ARRAYARRAY_UINT[1][7];

    RETAINTEST_AUTO_STRUCTUREARRAYARRAY.ARRAYARRAY_UINT[2][0] := RETAINTEST_AUTO_STRUCTUREARRAYARRAY.ARRAYARRAY_UINT[2][0] + 1;
    RETAINTEST_AUTO_STRUCTUREARRAYARRAY.ARRAYARRAY_UINT[2][1] := RETAINTEST_AUTO_STRUCTUREARRAYARRAY.ARRAYARRAY_UINT[2][1] + 1;
    RETAINTEST_AUTO_STRUCTUREARRAYARRAY.ARRAYARRAY_UINT[2][2] := RETAINTEST_AUTO_STRUCTUREARRAYARRAY.ARRAYARRAY_UINT[2][2] + 1;
    RETAINTEST_AUTO_STRUCTUREARRAYARRAY.ARRAYARRAY_UINT[2][3] := RETAINTEST_AUTO_STRUCTUREARRAYARRAY.ARRAYARRAY_UINT[2][3] + 1;
    RETAINTEST_AUTO_STRUCTUREARRAYARRAY.ARRAYARRAY_UINT[2][4] := RETAINTEST_AUTO_STRUCTUREARRAYARRAY.ARRAYARRAY_UINT[2][4] + 1;
    RETAINTEST_AUTO_STRUCTUREARRAYARRAY.ARRAYARRAY_UINT[2][5] := RETAINTEST_AUTO_STRUCTUREARRAYARRAY.ARRAYARRAY_UINT[2][5] + 1;
    RETAINTEST_AUTO_STRUCTUREARRAYARRAY.ARRAYARRAY_UINT[2][6] := RETAINTEST_AUTO_STRUCTUREARRAYARRAY.ARRAYARRAY_UINT[2][6] + 1;
    RETAINTEST_AUTO_STRUCTUREARRAYARRAY.ARRAYARRAY_UINT[2][7] := RETAINTEST_AUTO_STRUCTUREARRAYARRAY.ARRAYARRAY_UINT[2][7] + 1;
    RETAINTEST_AUTO_STRUCTUREARRAYARRAY.ARRAYARRAY_UINT[2][8] := RETAINTEST_AUTO_STRUCTUREARRAYARRAY.ARRAYARRAY_UINT[2][8] + 1;
    RETAINTEST_AUTO_STRUCTUREARRAYARRAY.ARRAYARRAY_UINT[2][9] := RETAINTEST_AUTO_STRUCTUREARRAYARRAY.ARRAYARRAY_UINT[2][9] + 1;

    RETAINTEST_AUTO_STRUCTUREARRAYARRAY.ARRAYARRAY_UINT[3][0] := RETAINTEST_AUTO_STRUCTUREARRAYARRAY.ARRAYARRAY_UINT[3][0] + 1;
    RETAINTEST_AUTO_STRUCTUREARRAYARRAY.ARRAYARRAY_UINT[3][1] := RETAINTEST_AUTO_STRUCTUREARRAYARRAY.ARRAYARRAY_UINT[3][1] + 1;
    RETAINTEST_AUTO_STRUCTUREARRAYARRAY.ARRAYARRAY_UINT[3][2] := RETAINTEST_AUTO_STRUCTUREARRAYARRAY.ARRAYARRAY_UINT[3][2] + 1;
    RETAINTEST_AUTO_STRUCTUREARRAYARRAY.ARRAYARRAY_UINT[3][3] := RETAINTEST_AUTO_STRUCTUREARRAYARRAY.ARRAYARRAY_UINT[3][3] + 1;
    RETAINTEST_AUTO_STRUCTUREARRAYARRAY.ARRAYARRAY_UINT[3][4] := RETAINTEST_AUTO_STRUCTUREARRAYARRAY.ARRAYARRAY_UINT[3][4] + 1;
    RETAINTEST_AUTO_STRUCTUREARRAYARRAY.ARRAYARRAY_UINT[3][5] := RETAINTEST_AUTO_STRUCTUREARRAYARRAY.ARRAYARRAY_UINT[3][5] + 1;
    RETAINTEST_AUTO_STRUCTUREARRAYARRAY.ARRAYARRAY_UINT[3][6] := RETAINTEST_AUTO_STRUCTUREARRAYARRAY.ARRAYARRAY_UINT[3][6] + 1;
    RETAINTEST_AUTO_STRUCTUREARRAYARRAY.ARRAYARRAY_UINT[3][7] := RETAINTEST_AUTO_STRUCTUREARRAYARRAY.ARRAYARRAY_UINT[3][7] + 1;
    RETAINTEST_AUTO_STRUCTUREARRAYARRAY.ARRAYARRAY_UINT[3][8] := RETAINTEST_AUTO_STRUCTUREARRAYARRAY.ARRAYARRAY_UINT[3][8] + 1;
    RETAINTEST_AUTO_STRUCTUREARRAYARRAY.ARRAYARRAY_UINT[3][9] := RETAINTEST_AUTO_STRUCTUREARRAYARRAY.ARRAYARRAY_UINT[3][9] + 1;

    RETAINTEST_AUTO_STRUCTUREARRAYARRAY.ARRAYARRAY_UINT[4][0] := RETAINTEST_AUTO_STRUCTUREARRAYARRAY.ARRAYARRAY_UINT[4][0] + 1;
    RETAINTEST_AUTO_STRUCTUREARRAYARRAY.ARRAYARRAY_UINT[4][1] := RETAINTEST_AUTO_STRUCTUREARRAYARRAY.ARRAYARRAY_UINT[4][1] + 1;
    RETAINTEST_AUTO_STRUCTUREARRAYARRAY.ARRAYARRAY_UINT[4][2] := RETAINTEST_AUTO_STRUCTUREARRAYARRAY.ARRAYARRAY_UINT[4][2] + 1;
    RETAINTEST_AUTO_STRUCTUREARRAYARRAY.ARRAYARRAY_UINT[4][3] := RETAINTEST_AUTO_STRUCTUREARRAYARRAY.ARRAYARRAY_UINT[4][3] + 1;
    RETAINTEST_AUTO_STRUCTUREARRAYARRAY.ARRAYARRAY_UINT[4][4] := RETAINTEST_AUTO_STRUCTUREARRAYARRAY.ARRAYARRAY_UINT[4][4] + 1;
    RETAINTEST_AUTO_STRUCTUREARRAYARRAY.ARRAYARRAY_UINT[4][5] := RETAINTEST_AUTO_STRUCTUREARRAYARRAY.ARRAYARRAY_UINT[4][5] + 1;
    RETAINTEST_AUTO_STRUCTUREARRAYARRAY.ARRAYARRAY_UINT[4][6] := RETAINTEST_AUTO_STRUCTUREARRAYARRAY.ARRAYARRAY_UINT[4][6] + 1;
    RETAINTEST_AUTO_STRUCTUREARRAYARRAY.ARRAYARRAY_UINT[4][7] := RETAINTEST_AUTO_STRUCTUREARRAYARRAY.ARRAYARRAY_UINT[4][7] + 1;
    RETAINTEST_AUTO_STRUCTUREARRAYARRAY.ARRAYARRAY_UINT[4][8] := RETAINTEST_AUTO_STRUCTUREARRAYARRAY.ARRAYARRAY_UINT[4][8] + 1;
    RETAINTEST_AUTO_STRUCTUREARRAYARRAY.ARRAYARRAY_UINT[4][9] := RETAINTEST_AUTO_STRUCTUREARRAYARRAY.ARRAYARRAY_UINT[4][9] + 1;

    RETAINTEST_AUTO_STRUCTUREARRAYARRAY.ARRAYARRAY_UINT[5][0] := RETAINTEST_AUTO_STRUCTUREARRAYARRAY.ARRAYARRAY_UINT[5][0] + 1;
    RETAINTEST_AUTO_STRUCTUREARRAYARRAY.ARRAYARRAY_UINT[5][1] := RETAINTEST_AUTO_STRUCTUREARRAYARRAY.ARRAYARRAY_UINT[5][1] + 1;
    RETAINTEST_AUTO_STRUCTUREARRAYARRAY.ARRAYARRAY_UINT[5][2] := RETAINTEST_AUTO_STRUCTUREARRAYARRAY.ARRAYARRAY_UINT[5][2] + 1;
    RETAINTEST_AUTO_STRUCTUREARRAYARRAY.ARRAYARRAY_UINT[5][3] := RETAINTEST_AUTO_STRUCTUREARRAYARRAY.ARRAYARRAY_UINT[5][3] + 1;
    RETAINTEST_AUTO_STRUCTUREARRAYARRAY.ARRAYARRAY_UINT[5][4] := RETAINTEST_AUTO_STRUCTUREARRAYARRAY.ARRAYARRAY_UINT[5][4] + 1;
    RETAINTEST_AUTO_STRUCTUREARRAYARRAY.ARRAYARRAY_UINT[5][5] := RETAINTEST_AUTO_STRUCTUREARRAYARRAY.ARRAYARRAY_UINT[5][5] + 1;
    RETAINTEST_AUTO_STRUCTUREARRAYARRAY.ARRAYARRAY_UINT[5][6] := RETAINTEST_AUTO_STRUCTUREARRAYARRAY.ARRAYARRAY_UINT[5][6] + 1;
    RETAINTEST_AUTO_STRUCTUREARRAYARRAY.ARRAYARRAY_UINT[5][7] := RETAINTEST_AUTO_STRUCTUREARRAYARRAY.ARRAYARRAY_UINT[5][7] + 1;
    RETAINTEST_AUTO_STRUCTUREARRAYARRAY.ARRAYARRAY_UINT[5][8] := RETAINTEST_AUTO_STRUCTUREARRAYARRAY.ARRAYARRAY_UINT[5][8] + 1;
    RETAINTEST_AUTO_STRUCTUREARRAYARRAY.ARRAYARRAY_UINT[5][9] := RETAINTEST_AUTO_STRUCTUREARRAYARRAY.ARRAYARRAY_UINT[5][9] + 1;

    RETAINTEST_AUTO_STRUCTUREARRAYARRAY.ARRAYARRAY_UINT[6][0] := RETAINTEST_AUTO_STRUCTUREARRAYARRAY.ARRAYARRAY_UINT[6][0] + 1;
    RETAINTEST_AUTO_STRUCTUREARRAYARRAY.ARRAYARRAY_UINT[6][1] := RETAINTEST_AUTO_STRUCTUREARRAYARRAY.ARRAYARRAY_UINT[6][1] + 1;
    RETAINTEST_AUTO_STRUCTUREARRAYARRAY.ARRAYARRAY_UINT[6][2] := RETAINTEST_AUTO_STRUCTUREARRAYARRAY.ARRAYARRAY_UINT[6][2] + 1;
    RETAINTEST_AUTO_STRUCTUREARRAYARRAY.ARRAYARRAY_UINT[6][3] := RETAINTEST_AUTO_STRUCTUREARRAYARRAY.ARRAYARRAY_UINT[6][3] + 1;
    RETAINTEST_AUTO_STRUCTUREARRAYARRAY.ARRAYARRAY_UINT[6][4] := RETAINTEST_AUTO_STRUCTUREARRAYARRAY.ARRAYARRAY_UINT[6][4] + 1;
    RETAINTEST_AUTO_STRUCTUREARRAYARRAY.ARRAYARRAY_UINT[6][5] := RETAINTEST_AUTO_STRUCTUREARRAYARRAY.ARRAYARRAY_UINT[6][5] + 1;
    RETAINTEST_AUTO_STRUCTUREARRAYARRAY.ARRAYARRAY_UINT[6][6] := RETAINTEST_AUTO_STRUCTUREARRAYARRAY.ARRAYARRAY_UINT[6][6] + 1;
    RETAINTEST_AUTO_STRUCTUREARRAYARRAY.ARRAYARRAY_UINT[6][7] := RETAINTEST_AUTO_STRUCTUREARRAYARRAY.ARRAYARRAY_UINT[6][7] + 1;
    RETAINTEST_AUTO_STRUCTUREARRAYARRAY.ARRAYARRAY_UINT[6][8] := RETAINTEST_AUTO_STRUCTUREARRAYARRAY.ARRAYARRAY_UINT[6][8] + 1;
    RETAINTEST_AUTO_STRUCTUREARRAYARRAY.ARRAYARRAY_UINT[6][9] := RETAINTEST_AUTO_STRUCTUREARRAYARRAY.ARRAYARRAY_UINT[6][9] + 1;

    RETAINTEST_AUTO_STRUCTUREARRAYARRAY.ARRAYARRAY_UINT[7][0] := RETAINTEST_AUTO_STRUCTUREARRAYARRAY.ARRAYARRAY_UINT[6][0];
    RETAINTEST_AUTO_STRUCTUREARRAYARRAY.ARRAYARRAY_UINT[7][1] := RETAINTEST_AUTO_STRUCTUREARRAYARRAY.ARRAYARRAY_UINT[6][1];
    RETAINTEST_AUTO_STRUCTUREARRAYARRAY.ARRAYARRAY_UINT[7][2] := RETAINTEST_AUTO_STRUCTUREARRAYARRAY.ARRAYARRAY_UINT[6][2];
    RETAINTEST_AUTO_STRUCTUREARRAYARRAY.ARRAYARRAY_UINT[7][3] := RETAINTEST_AUTO_STRUCTUREARRAYARRAY.ARRAYARRAY_UINT[6][3];
    RETAINTEST_AUTO_STRUCTUREARRAYARRAY.ARRAYARRAY_UINT[7][4] := RETAINTEST_AUTO_STRUCTUREARRAYARRAY.ARRAYARRAY_UINT[6][4];
    RETAINTEST_AUTO_STRUCTUREARRAYARRAY.ARRAYARRAY_UINT[7][5] := RETAINTEST_AUTO_STRUCTUREARRAYARRAY.ARRAYARRAY_UINT[6][5];
    RETAINTEST_AUTO_STRUCTUREARRAYARRAY.ARRAYARRAY_UINT[7][6] := RETAINTEST_AUTO_STRUCTUREARRAYARRAY.ARRAYARRAY_UINT[6][6];
    RETAINTEST_AUTO_STRUCTUREARRAYARRAY.ARRAYARRAY_UINT[7][7] := RETAINTEST_AUTO_STRUCTUREARRAYARRAY.ARRAYARRAY_UINT[6][7];
    RETAINTEST_AUTO_STRUCTUREARRAYARRAY.ARRAYARRAY_UINT[7][8] := RETAINTEST_AUTO_STRUCTUREARRAYARRAY.ARRAYARRAY_UINT[6][8];
    RETAINTEST_AUTO_STRUCTUREARRAYARRAY.ARRAYARRAY_UINT[7][9] := RETAINTEST_AUTO_STRUCTUREARRAYARRAY.ARRAYARRAY_UINT[6][9];

    RETAINTEST_AUTO_STRUCTUREARRAYARRAY.ARRAYARRAY_ULINT[0][0] := RETAINTEST_AUTO_STRUCTUREARRAYARRAY.ARRAYARRAY_ULINT[0][0] + 1;
    RETAINTEST_AUTO_STRUCTUREARRAYARRAY.ARRAYARRAY_ULINT[0][1] := RETAINTEST_AUTO_STRUCTUREARRAYARRAY.ARRAYARRAY_ULINT[0][1] + 1;
    RETAINTEST_AUTO_STRUCTUREARRAYARRAY.ARRAYARRAY_ULINT[0][2] := RETAINTEST_AUTO_STRUCTUREARRAYARRAY.ARRAYARRAY_ULINT[0][2] + 1;
    RETAINTEST_AUTO_STRUCTUREARRAYARRAY.ARRAYARRAY_ULINT[0][3] := RETAINTEST_AUTO_STRUCTUREARRAYARRAY.ARRAYARRAY_ULINT[0][3] + 1;
    RETAINTEST_AUTO_STRUCTUREARRAYARRAY.ARRAYARRAY_ULINT[0][4] := RETAINTEST_AUTO_STRUCTUREARRAYARRAY.ARRAYARRAY_ULINT[0][4] + 1;
    RETAINTEST_AUTO_STRUCTUREARRAYARRAY.ARRAYARRAY_ULINT[0][5] := RETAINTEST_AUTO_STRUCTUREARRAYARRAY.ARRAYARRAY_ULINT[0][5] + 1;
    RETAINTEST_AUTO_STRUCTUREARRAYARRAY.ARRAYARRAY_ULINT[0][6] := RETAINTEST_AUTO_STRUCTUREARRAYARRAY.ARRAYARRAY_ULINT[0][6] + 1;
    RETAINTEST_AUTO_STRUCTUREARRAYARRAY.ARRAYARRAY_ULINT[0][7] := RETAINTEST_AUTO_STRUCTUREARRAYARRAY.ARRAYARRAY_ULINT[0][7] + 1;
    RETAINTEST_AUTO_STRUCTUREARRAYARRAY.ARRAYARRAY_ULINT[0][8] := RETAINTEST_AUTO_STRUCTUREARRAYARRAY.ARRAYARRAY_ULINT[0][6];
    RETAINTEST_AUTO_STRUCTUREARRAYARRAY.ARRAYARRAY_ULINT[0][9] := RETAINTEST_AUTO_STRUCTUREARRAYARRAY.ARRAYARRAY_ULINT[0][7];

    RETAINTEST_AUTO_STRUCTUREARRAYARRAY.ARRAYARRAY_ULINT[1][0] := RETAINTEST_AUTO_STRUCTUREARRAYARRAY.ARRAYARRAY_ULINT[1][0] + 1;
    RETAINTEST_AUTO_STRUCTUREARRAYARRAY.ARRAYARRAY_ULINT[1][1] := RETAINTEST_AUTO_STRUCTUREARRAYARRAY.ARRAYARRAY_ULINT[1][1] + 1;
    RETAINTEST_AUTO_STRUCTUREARRAYARRAY.ARRAYARRAY_ULINT[1][2] := RETAINTEST_AUTO_STRUCTUREARRAYARRAY.ARRAYARRAY_ULINT[1][2] + 1;
    RETAINTEST_AUTO_STRUCTUREARRAYARRAY.ARRAYARRAY_ULINT[1][3] := RETAINTEST_AUTO_STRUCTUREARRAYARRAY.ARRAYARRAY_ULINT[1][3] + 1;
    RETAINTEST_AUTO_STRUCTUREARRAYARRAY.ARRAYARRAY_ULINT[1][4] := RETAINTEST_AUTO_STRUCTUREARRAYARRAY.ARRAYARRAY_ULINT[1][4] + 1;
    RETAINTEST_AUTO_STRUCTUREARRAYARRAY.ARRAYARRAY_ULINT[1][5] := RETAINTEST_AUTO_STRUCTUREARRAYARRAY.ARRAYARRAY_ULINT[1][5] + 1;
    RETAINTEST_AUTO_STRUCTUREARRAYARRAY.ARRAYARRAY_ULINT[1][6] := RETAINTEST_AUTO_STRUCTUREARRAYARRAY.ARRAYARRAY_ULINT[1][6] + 1;
    RETAINTEST_AUTO_STRUCTUREARRAYARRAY.ARRAYARRAY_ULINT[1][7] := RETAINTEST_AUTO_STRUCTUREARRAYARRAY.ARRAYARRAY_ULINT[1][7] + 1;
    RETAINTEST_AUTO_STRUCTUREARRAYARRAY.ARRAYARRAY_ULINT[1][8] := RETAINTEST_AUTO_STRUCTUREARRAYARRAY.ARRAYARRAY_ULINT[1][6];
    RETAINTEST_AUTO_STRUCTUREARRAYARRAY.ARRAYARRAY_ULINT[1][9] := RETAINTEST_AUTO_STRUCTUREARRAYARRAY.ARRAYARRAY_ULINT[1][7];

    RETAINTEST_AUTO_STRUCTUREARRAYARRAY.ARRAYARRAY_ULINT[2][0] := RETAINTEST_AUTO_STRUCTUREARRAYARRAY.ARRAYARRAY_ULINT[2][0] + 1;
    RETAINTEST_AUTO_STRUCTUREARRAYARRAY.ARRAYARRAY_ULINT[2][1] := RETAINTEST_AUTO_STRUCTUREARRAYARRAY.ARRAYARRAY_ULINT[2][1] + 1;
    RETAINTEST_AUTO_STRUCTUREARRAYARRAY.ARRAYARRAY_ULINT[2][2] := RETAINTEST_AUTO_STRUCTUREARRAYARRAY.ARRAYARRAY_ULINT[2][2] + 1;
    RETAINTEST_AUTO_STRUCTUREARRAYARRAY.ARRAYARRAY_ULINT[2][3] := RETAINTEST_AUTO_STRUCTUREARRAYARRAY.ARRAYARRAY_ULINT[2][3] + 1;
    RETAINTEST_AUTO_STRUCTUREARRAYARRAY.ARRAYARRAY_ULINT[2][4] := RETAINTEST_AUTO_STRUCTUREARRAYARRAY.ARRAYARRAY_ULINT[2][4] + 1;
    RETAINTEST_AUTO_STRUCTUREARRAYARRAY.ARRAYARRAY_ULINT[2][5] := RETAINTEST_AUTO_STRUCTUREARRAYARRAY.ARRAYARRAY_ULINT[2][5] + 1;
    RETAINTEST_AUTO_STRUCTUREARRAYARRAY.ARRAYARRAY_ULINT[2][6] := RETAINTEST_AUTO_STRUCTUREARRAYARRAY.ARRAYARRAY_ULINT[2][6] + 1;
    RETAINTEST_AUTO_STRUCTUREARRAYARRAY.ARRAYARRAY_ULINT[2][7] := RETAINTEST_AUTO_STRUCTUREARRAYARRAY.ARRAYARRAY_ULINT[2][7] + 1;
    RETAINTEST_AUTO_STRUCTUREARRAYARRAY.ARRAYARRAY_ULINT[2][8] := RETAINTEST_AUTO_STRUCTUREARRAYARRAY.ARRAYARRAY_ULINT[2][8] + 1;
    RETAINTEST_AUTO_STRUCTUREARRAYARRAY.ARRAYARRAY_ULINT[2][9] := RETAINTEST_AUTO_STRUCTUREARRAYARRAY.ARRAYARRAY_ULINT[2][9] + 1;

    RETAINTEST_AUTO_STRUCTUREARRAYARRAY.ARRAYARRAY_ULINT[3][0] := RETAINTEST_AUTO_STRUCTUREARRAYARRAY.ARRAYARRAY_ULINT[3][0] + 1;
    RETAINTEST_AUTO_STRUCTUREARRAYARRAY.ARRAYARRAY_ULINT[3][1] := RETAINTEST_AUTO_STRUCTUREARRAYARRAY.ARRAYARRAY_ULINT[3][1] + 1;
    RETAINTEST_AUTO_STRUCTUREARRAYARRAY.ARRAYARRAY_ULINT[3][2] := RETAINTEST_AUTO_STRUCTUREARRAYARRAY.ARRAYARRAY_ULINT[3][2] + 1;
    RETAINTEST_AUTO_STRUCTUREARRAYARRAY.ARRAYARRAY_ULINT[3][3] := RETAINTEST_AUTO_STRUCTUREARRAYARRAY.ARRAYARRAY_ULINT[3][3] + 1;
    RETAINTEST_AUTO_STRUCTUREARRAYARRAY.ARRAYARRAY_ULINT[3][4] := RETAINTEST_AUTO_STRUCTUREARRAYARRAY.ARRAYARRAY_ULINT[3][4] + 1;
    RETAINTEST_AUTO_STRUCTUREARRAYARRAY.ARRAYARRAY_ULINT[3][5] := RETAINTEST_AUTO_STRUCTUREARRAYARRAY.ARRAYARRAY_ULINT[3][5] + 1;
    RETAINTEST_AUTO_STRUCTUREARRAYARRAY.ARRAYARRAY_ULINT[3][6] := RETAINTEST_AUTO_STRUCTUREARRAYARRAY.ARRAYARRAY_ULINT[3][6] + 1;
    RETAINTEST_AUTO_STRUCTUREARRAYARRAY.ARRAYARRAY_ULINT[3][7] := RETAINTEST_AUTO_STRUCTUREARRAYARRAY.ARRAYARRAY_ULINT[3][7] + 1;
    RETAINTEST_AUTO_STRUCTUREARRAYARRAY.ARRAYARRAY_ULINT[3][8] := RETAINTEST_AUTO_STRUCTUREARRAYARRAY.ARRAYARRAY_ULINT[3][8] + 1;
    RETAINTEST_AUTO_STRUCTUREARRAYARRAY.ARRAYARRAY_ULINT[3][9] := RETAINTEST_AUTO_STRUCTUREARRAYARRAY.ARRAYARRAY_ULINT[3][9] + 1;

    RETAINTEST_AUTO_STRUCTUREARRAYARRAY.ARRAYARRAY_ULINT[4][0] := RETAINTEST_AUTO_STRUCTUREARRAYARRAY.ARRAYARRAY_ULINT[4][0] + 1;
    RETAINTEST_AUTO_STRUCTUREARRAYARRAY.ARRAYARRAY_ULINT[4][1] := RETAINTEST_AUTO_STRUCTUREARRAYARRAY.ARRAYARRAY_ULINT[4][1] + 1;
    RETAINTEST_AUTO_STRUCTUREARRAYARRAY.ARRAYARRAY_ULINT[4][2] := RETAINTEST_AUTO_STRUCTUREARRAYARRAY.ARRAYARRAY_ULINT[4][2] + 1;
    RETAINTEST_AUTO_STRUCTUREARRAYARRAY.ARRAYARRAY_ULINT[4][3] := RETAINTEST_AUTO_STRUCTUREARRAYARRAY.ARRAYARRAY_ULINT[4][3] + 1;
    RETAINTEST_AUTO_STRUCTUREARRAYARRAY.ARRAYARRAY_ULINT[4][4] := RETAINTEST_AUTO_STRUCTUREARRAYARRAY.ARRAYARRAY_ULINT[4][4] + 1;
    RETAINTEST_AUTO_STRUCTUREARRAYARRAY.ARRAYARRAY_ULINT[4][5] := RETAINTEST_AUTO_STRUCTUREARRAYARRAY.ARRAYARRAY_ULINT[4][5] + 1;
    RETAINTEST_AUTO_STRUCTUREARRAYARRAY.ARRAYARRAY_ULINT[4][6] := RETAINTEST_AUTO_STRUCTUREARRAYARRAY.ARRAYARRAY_ULINT[4][6] + 1;
    RETAINTEST_AUTO_STRUCTUREARRAYARRAY.ARRAYARRAY_ULINT[4][7] := RETAINTEST_AUTO_STRUCTUREARRAYARRAY.ARRAYARRAY_ULINT[4][7] + 1;
    RETAINTEST_AUTO_STRUCTUREARRAYARRAY.ARRAYARRAY_ULINT[4][8] := RETAINTEST_AUTO_STRUCTUREARRAYARRAY.ARRAYARRAY_ULINT[4][8] + 1;
    RETAINTEST_AUTO_STRUCTUREARRAYARRAY.ARRAYARRAY_ULINT[4][9] := RETAINTEST_AUTO_STRUCTUREARRAYARRAY.ARRAYARRAY_ULINT[4][9] + 1;

    RETAINTEST_AUTO_STRUCTUREARRAYARRAY.ARRAYARRAY_ULINT[5][0] := RETAINTEST_AUTO_STRUCTUREARRAYARRAY.ARRAYARRAY_ULINT[5][0] + 1;
    RETAINTEST_AUTO_STRUCTUREARRAYARRAY.ARRAYARRAY_ULINT[5][1] := RETAINTEST_AUTO_STRUCTUREARRAYARRAY.ARRAYARRAY_ULINT[5][1] + 1;
    RETAINTEST_AUTO_STRUCTUREARRAYARRAY.ARRAYARRAY_ULINT[5][2] := RETAINTEST_AUTO_STRUCTUREARRAYARRAY.ARRAYARRAY_ULINT[5][2] + 1;
    RETAINTEST_AUTO_STRUCTUREARRAYARRAY.ARRAYARRAY_ULINT[5][3] := RETAINTEST_AUTO_STRUCTUREARRAYARRAY.ARRAYARRAY_ULINT[5][3] + 1;
    RETAINTEST_AUTO_STRUCTUREARRAYARRAY.ARRAYARRAY_ULINT[5][4] := RETAINTEST_AUTO_STRUCTUREARRAYARRAY.ARRAYARRAY_ULINT[5][4] + 1;
    RETAINTEST_AUTO_STRUCTUREARRAYARRAY.ARRAYARRAY_ULINT[5][5] := RETAINTEST_AUTO_STRUCTUREARRAYARRAY.ARRAYARRAY_ULINT[5][5] + 1;
    RETAINTEST_AUTO_STRUCTUREARRAYARRAY.ARRAYARRAY_ULINT[5][6] := RETAINTEST_AUTO_STRUCTUREARRAYARRAY.ARRAYARRAY_ULINT[5][6] + 1;
    RETAINTEST_AUTO_STRUCTUREARRAYARRAY.ARRAYARRAY_ULINT[5][7] := RETAINTEST_AUTO_STRUCTUREARRAYARRAY.ARRAYARRAY_ULINT[5][7] + 1;
    RETAINTEST_AUTO_STRUCTUREARRAYARRAY.ARRAYARRAY_ULINT[5][8] := RETAINTEST_AUTO_STRUCTUREARRAYARRAY.ARRAYARRAY_ULINT[5][8] + 1;
    RETAINTEST_AUTO_STRUCTUREARRAYARRAY.ARRAYARRAY_ULINT[5][9] := RETAINTEST_AUTO_STRUCTUREARRAYARRAY.ARRAYARRAY_ULINT[5][9] + 1;

    RETAINTEST_AUTO_STRUCTUREARRAYARRAY.ARRAYARRAY_ULINT[6][0] := RETAINTEST_AUTO_STRUCTUREARRAYARRAY.ARRAYARRAY_ULINT[6][0] + 1;
    RETAINTEST_AUTO_STRUCTUREARRAYARRAY.ARRAYARRAY_ULINT[6][1] := RETAINTEST_AUTO_STRUCTUREARRAYARRAY.ARRAYARRAY_ULINT[6][1] + 1;
    RETAINTEST_AUTO_STRUCTUREARRAYARRAY.ARRAYARRAY_ULINT[6][2] := RETAINTEST_AUTO_STRUCTUREARRAYARRAY.ARRAYARRAY_ULINT[6][2] + 1;
    RETAINTEST_AUTO_STRUCTUREARRAYARRAY.ARRAYARRAY_ULINT[6][3] := RETAINTEST_AUTO_STRUCTUREARRAYARRAY.ARRAYARRAY_ULINT[6][3] + 1;
    RETAINTEST_AUTO_STRUCTUREARRAYARRAY.ARRAYARRAY_ULINT[6][4] := RETAINTEST_AUTO_STRUCTUREARRAYARRAY.ARRAYARRAY_ULINT[6][4] + 1;
    RETAINTEST_AUTO_STRUCTUREARRAYARRAY.ARRAYARRAY_ULINT[6][5] := RETAINTEST_AUTO_STRUCTUREARRAYARRAY.ARRAYARRAY_ULINT[6][5] + 1;
    RETAINTEST_AUTO_STRUCTUREARRAYARRAY.ARRAYARRAY_ULINT[6][6] := RETAINTEST_AUTO_STRUCTUREARRAYARRAY.ARRAYARRAY_ULINT[6][6] + 1;
    RETAINTEST_AUTO_STRUCTUREARRAYARRAY.ARRAYARRAY_ULINT[6][7] := RETAINTEST_AUTO_STRUCTUREARRAYARRAY.ARRAYARRAY_ULINT[6][7] + 1;
    RETAINTEST_AUTO_STRUCTUREARRAYARRAY.ARRAYARRAY_ULINT[6][8] := RETAINTEST_AUTO_STRUCTUREARRAYARRAY.ARRAYARRAY_ULINT[6][8] + 1;
    RETAINTEST_AUTO_STRUCTUREARRAYARRAY.ARRAYARRAY_ULINT[6][9] := RETAINTEST_AUTO_STRUCTUREARRAYARRAY.ARRAYARRAY_ULINT[6][9] + 1;

    RETAINTEST_AUTO_STRUCTUREARRAYARRAY.ARRAYARRAY_ULINT[7][0] := RETAINTEST_AUTO_STRUCTUREARRAYARRAY.ARRAYARRAY_ULINT[6][0];
    RETAINTEST_AUTO_STRUCTUREARRAYARRAY.ARRAYARRAY_ULINT[7][1] := RETAINTEST_AUTO_STRUCTUREARRAYARRAY.ARRAYARRAY_ULINT[6][1];
    RETAINTEST_AUTO_STRUCTUREARRAYARRAY.ARRAYARRAY_ULINT[7][2] := RETAINTEST_AUTO_STRUCTUREARRAYARRAY.ARRAYARRAY_ULINT[6][2];
    RETAINTEST_AUTO_STRUCTUREARRAYARRAY.ARRAYARRAY_ULINT[7][3] := RETAINTEST_AUTO_STRUCTUREARRAYARRAY.ARRAYARRAY_ULINT[6][3];
    RETAINTEST_AUTO_STRUCTUREARRAYARRAY.ARRAYARRAY_ULINT[7][4] := RETAINTEST_AUTO_STRUCTUREARRAYARRAY.ARRAYARRAY_ULINT[6][4];
    RETAINTEST_AUTO_STRUCTUREARRAYARRAY.ARRAYARRAY_ULINT[7][5] := RETAINTEST_AUTO_STRUCTUREARRAYARRAY.ARRAYARRAY_ULINT[6][5];
    RETAINTEST_AUTO_STRUCTUREARRAYARRAY.ARRAYARRAY_ULINT[7][6] := RETAINTEST_AUTO_STRUCTUREARRAYARRAY.ARRAYARRAY_ULINT[6][6];
    RETAINTEST_AUTO_STRUCTUREARRAYARRAY.ARRAYARRAY_ULINT[7][7] := RETAINTEST_AUTO_STRUCTUREARRAYARRAY.ARRAYARRAY_ULINT[6][7];
    RETAINTEST_AUTO_STRUCTUREARRAYARRAY.ARRAYARRAY_ULINT[7][8] := RETAINTEST_AUTO_STRUCTUREARRAYARRAY.ARRAYARRAY_ULINT[6][8];
    RETAINTEST_AUTO_STRUCTUREARRAYARRAY.ARRAYARRAY_ULINT[7][9] := RETAINTEST_AUTO_STRUCTUREARRAYARRAY.ARRAYARRAY_ULINT[6][9];

    RETAINTEST_AUTO_STRUCTUREARRAYARRAY.ARRAYARRAY_USINT[0][0] := RETAINTEST_AUTO_STRUCTUREARRAYARRAY.ARRAYARRAY_USINT[0][0] + 1;
    RETAINTEST_AUTO_STRUCTUREARRAYARRAY.ARRAYARRAY_USINT[0][1] := RETAINTEST_AUTO_STRUCTUREARRAYARRAY.ARRAYARRAY_USINT[0][1] + 1;
    RETAINTEST_AUTO_STRUCTUREARRAYARRAY.ARRAYARRAY_USINT[0][2] := RETAINTEST_AUTO_STRUCTUREARRAYARRAY.ARRAYARRAY_USINT[0][2] + 1;
    RETAINTEST_AUTO_STRUCTUREARRAYARRAY.ARRAYARRAY_USINT[0][3] := RETAINTEST_AUTO_STRUCTUREARRAYARRAY.ARRAYARRAY_USINT[0][3] + 1;
    RETAINTEST_AUTO_STRUCTUREARRAYARRAY.ARRAYARRAY_USINT[0][4] := RETAINTEST_AUTO_STRUCTUREARRAYARRAY.ARRAYARRAY_USINT[0][4] + 1;
    RETAINTEST_AUTO_STRUCTUREARRAYARRAY.ARRAYARRAY_USINT[0][5] := RETAINTEST_AUTO_STRUCTUREARRAYARRAY.ARRAYARRAY_USINT[0][5] + 1;
    RETAINTEST_AUTO_STRUCTUREARRAYARRAY.ARRAYARRAY_USINT[0][6] := RETAINTEST_AUTO_STRUCTUREARRAYARRAY.ARRAYARRAY_USINT[0][6] + 1;
    RETAINTEST_AUTO_STRUCTUREARRAYARRAY.ARRAYARRAY_USINT[0][7] := RETAINTEST_AUTO_STRUCTUREARRAYARRAY.ARRAYARRAY_USINT[0][7] + 1;
    RETAINTEST_AUTO_STRUCTUREARRAYARRAY.ARRAYARRAY_USINT[0][8] := RETAINTEST_AUTO_STRUCTUREARRAYARRAY.ARRAYARRAY_USINT[0][6];
    RETAINTEST_AUTO_STRUCTUREARRAYARRAY.ARRAYARRAY_USINT[0][9] := RETAINTEST_AUTO_STRUCTUREARRAYARRAY.ARRAYARRAY_USINT[0][7];
